(* CoDeSys 2.3 export: OSCAT260.TXT *)
(* Libraries: STANDARD.LIB 4.10.05 11:14:46 *)

(* Global variable list: Constants *)
VAR_GLOBAL CONSTANT
	(* setup Parameters *)
	STEP7 : BOOL := FALSE;

	(* Mathematische Konstanten *)
	PI1 : REAL := 3.14159265358979323846264338327950288;	(* Kreiszahl PI *)
	PI2 : REAL := 6.283185307179586476;					(* PI * 2 *)
	E : REAL := 2.71828182845904523536028747135266249;	(* Eulersche Konstante *)

	(* Physikalische Konstanten *)
	C0 : REAL := 299792458 ;							(* Lichtgeschwindigkeit in m/s *)
	EL : REAL := 1.60217653E-19;						(* elementarladung in Colomb = A * s *)
	GN : REAL := 9.80665; 								(* Erdbeschleunigung in m / s² *)
	TK : REAL := -273.15;									(* absoluter Nullpunkt in °C *)
	RU : REAL := 8.314472; 								(*Universelle Gaskonstante in J / (mol · K) *)
	PN : REAL := 101325;									(* NormalDruck in Pa *)

END_VAR

VAR_GLOBAL
END_VAR

(* revisionhistory
hm 3.3.2007
	extended accuracy of pi2
	renamed T0 to Tk for better compatibility with other libraries
	renamed C t0 c0 for better compatibility

hm	2.5.2007
	added RU universal gas constant

hm	1. oct 2007
	added setup parameter STEP7

hm 31. oct 2007
	added PN
*)

(* Data type *)
TYPE esr_data :
STRUCT
	typ : BYTE;
	adress : STRING(10);
	DS : DT;
	TS : TIME;
	data : ARRAY[0..7] OF BYTE;
END_STRUCT
END_TYPE

(* Data type *)
TYPE vector_3 :
STRUCT
	X : REAL;
	Y : REAL;
	Z : REAL;
END_STRUCT
END_TYPE

(* POU Building/actuators/actuator_2P, ST *)
FUNCTION_BLOCK actuator_2P
VAR_INPUT
	val : REAL;
	force : BOOL;
	force_in : BOOL;
END_VAR
VAR_INPUT CONSTANT
	self_act_time : TIME := t#10d;
	self_act_cycles : INT := 5;
	cycle_time : TIME := t#10m;
	min_ontime : TIME := t#10s;
	min_offtime : TIME := t#10s;
END_VAR
VAR_OUTPUT
	out :BOOL;
	pos : REAL;
END_VAR
VAR
	last_activation : TIME;
	count : INT;
	TON : TIME;
	tx : TIME;
	tc : TIME;
END_VAR


(*
version 1.5	27 dec 2007
programmer 	hugo
tested by		tobias

this is an intelligent actuator interface for any 2point actuator like coil drive.
the 2Point actuator can only switch on/off and therefore a input must be converted to on/off cycles.
the interface can be programmed with double click on the symbol for duty cyle, min_ontime and min_offtime to avoid flickering of the valve or flap.
in addition a self_act_time and self_act_cycles ca be programmed to switch n times on/off every self_act_time to avoid a valve to freeze.
a on and off input can be used to force the valve on or off at all times.
a additional pos output will always indicate the current position of a valve.
the input value must be between 0 and 1.

val		force	force_in	pos	out			
X		0		-			X		duty cycle X
-		1		1			1		1
-		1		0			0		0

*)
(* read system Time *)
tx := DWORD_TO_TIME(T_PLC_MS());
tc := tx - last_activation;

(* verify input to be between 0 and 1 *)
val := LIMIT(0,val,1);

(* check for min ontime or min offtime and wait if not passed *)
IF (out AND tc < min_ontime) OR (NOT out AND tc < min_offtime) THEN RETURN;

(* when force off then shutoff valve *)
ELSIF force AND NOT force_in THEN
	pos := 0;
	out := 0;
	last_activation := tx;
	count := 0;

(* if force on then turn on valve *)

ELSIF force AND force_in THEN
	pos := 1;
	out := 1;
	last_activation := tx;
	count := 0;

(* if nothing happened for self_act_time then do self activation cycles *)
ELSIF (tc >= self_act_time AND count = 0 AND self_act_cycles > 0) OR (count > 0 AND count < self_act_cycles * 2) THEN
	out := NOT out;
	last_activation := tx;
	count := count + 1;
	RETURN;
ELSIF count > 0 THEN
	count := 0;
ELSE
	ton := multime(cycle_time,val);
	IF ton < min_ontime / 2 THEN ton := t#0s; ELSIF ton < min_ontime THEN ton := min_ontime; END_IF;
	IF ton > cycle_time - min_offtime / 2 THEN ton := cycle_time; ELSIF ton > cycle_time - min_offtime THEN ton := cycle_time - min_offtime; END_IF;
	IF ton = t#0s THEN
		IF out =0 THEN
			pos := 0;
			RETURN;
		ELSE
			out := 0;
			pos := 0;
			last_activation := tx;
		END_IF;
	ELSIF ton = cycle_time THEN
		IF out = 1 THEN
			pos := 1;
			RETURN;
		ELSE
			out := 1;
			pos := 1;
			last_activation := tx;
		END_IF;
	END_IF;
	pos := TIME_TO_REAL(ton) / TIME_TO_REAL(cycle_time);
	(* output pulse generation *)
	IF out AND tc >= ton THEN
		out := 0;
		last_activation := tx;
	ELSIF NOT out AND tc >= cycle_time - ton THEN
		out := 1;
		last_activation := tx;
	END_IF;
END_IF;


(*
revision history:

hm		7.10.2006 		rev 1.1
	changed error pos could not reach 1 or 0 under certain conditions due to error in code.
	changed on and off in force and force_in for better usability.

hm		17.1.2007		rev 1.2
	deleted unused variable time_overflow

hm		15.9.2007		rev 1.3
	replaced time() with T_PLC_MS for compatibility and performance reasons

hm		19. 11 2007		rev 1.4
	replaced left over statement time() with tx

hm		27. 12. 2007	REV 1.5
	CHANGED CODE FOR BETTER PERFORMANCE
*)
END_FUNCTION_BLOCK

(* POU engineering/measurements/cycle_time, ST *)
FUNCTION_BLOCK cycle_time
VAR_INPUT
	rst : BOOL;
END_VAR
VAR_OUTPUT
	ct_min : TIME := t#0s;
	ct_max : TIME := t#0s;
	ct_last : TIME;
	systime : TIME;
	sysdays : INT;
	cycles : DWORD;
END_VAR
VAR
	last_cycle : TIME;
	tx: TIME;
	init: BOOL;
END_VAR


(*
	version 1.2	16 sep 2007
	programmer 	hugo
	tested BY		hans

this function block measures the cycle time and displays the last, min and max cycle time of the current task.
the resolution is 1ms.
the cycles output is a dword counter which counts the cycles.
a rst pulse on the input will reset all data.


*)
tx := DWORD_TO_TIME(T_PLC_MS()) - last_cycle;
IF rst THEN
	ct_min := t#10h;
	ct_max := t#0ms;
	cycles := 0;
ELSIF last_cycle > t#0s THEN
	IF tx < ct_min THEN ct_min := tx;
	ELSIF tx > ct_max THEN ct_max := tx;
	END_IF;
	ct_last := tx;
ELSIF ct_min = t#0s THEN
	ct_min := t#0s - t#1ms;
END_IF;
IF init THEN
	systime := systime + tx;
		IF systime >= t#1d THEN
			systime := systime - t#1d;
			sysdays := sysdays + 1;
		END_IF;
END_IF;
init := TRUE;
last_cycle := last_cycle + tx;
cycles := cycles + 1;

(*	revision history
hm 12.12.2006		rev 1.1
	added cycles output, a dword cycle counter.
hm 10.3.2007			rev 1.2
	changed initialization of ct_min to t#10h for compatibility with siemens s7

hm	16.9.2007		rev 1.2
	changed Time() in T_PLC_MS() for compatibility resons

*)
END_FUNCTION_BLOCK

(* POU engineering/measurements/T_PLC_MS, ST *)
FUNCTION T_PLC_MS : DWORD
VAR CONSTANT
	debug : BOOL := FALSE;
	N : INT := 0;
	offset : DWORD := 0;
END_VAR
VAR
	tx : TIME;
	temp : DWORD := 1;
END_VAR

(*
version 1.1	12 nov 2007
programmer 	hugo
tested by		tobias

T_PLC_MS reads the internal PLC timer and return the time, it has the advantage to be able to set a debug mode 
and speed up the counter to test the plc timer overrun which occurs every 50 days respectively 25 days at siemens S7
this routine also allows to correct the behavior of s7 where the internal plc counter will not count all 32 bits.

*)
tx := TIME();
T_PLC_MS := TIME_TO_DWORD(Tx);
(* hier muss die korrektur für step7 stattfinden
plctime muss den vollen wertebereich von time ausnutzen:
wenn bei step7 time -24tage bis plus 24 tage ist dann muss der timer auch beim überlauf auf -24tage springen 
und auf keinen fall auf 0 !!!!
für siemens muss ein weiterer fb im main eingebunden werden der sicherstellt das alle 32 bits durchgezählt werden.
es kann nur ein fb sein den er muss sich das oberste (32te) bit merken.
oder etwa spring s7 bei überlauf auf -24 tage????? dann wäre keine korrektur nötig.
*)
IF debug THEN
	T_PLC_MS := (SHL(T_PLC_MS,N) OR SHL(temp,N)-1) + Offset;
END_IF;

(* revision history
hm	14.9.2007	rev 1.0
	original version

hm	12. nov 2007	rev 1.1
	added temporaray variable tx because some compilers could not handle time() as an argument

*)
END_FUNCTION

(* POU engineering/signal processing/Offset, ST *)
FUNCTION Offset : REAL
VAR_INPUT
	X : REAL;
	O1, O2, O3, O4 : BOOL;
	D : BOOL;
END_VAR
VAR_INPUT CONSTANT
	Offset_1 : REAL;
	Offset_2 : REAL;
	Offset_3 : REAL;
	Offset_4 : REAL;
	default : REAL;
END_VAR

(*
version 1.0	12 jan 2007
programmer 	oscat
tested by		tobias

The Function offset adds offsets to an analog signal depending on digital inputs.
all selected offsets are added at the same time.
with the input D a default value instead of the input X can be used.

*) 
IF D THEN Offset := default; ELSE Offset := X; END_IF;
IF O1 THEN Offset := Offset + offset_1; END_IF;
IF O2 THEN Offset := Offset + offset_2; END_IF;
IF O3 THEN Offset := Offset + offset_3; END_IF;
IF O4 THEN Offset := Offset + offset_4; END_IF;
END_FUNCTION

(* POU Time&Date/multime, ST *)
FUNCTION multime : TIME
VAR_INPUT
	t : TIME;
	M : REAL;
END_VAR
VAR
END_VAR


(*
version 1.0	2 oct 2006
programmer 	hugo
tested by		tobias

multiplies a time by a real number and returns a time
*)
multime := REAL_TO_TIME(TIME_TO_REAL(t)*M);
END_FUNCTION

(* POU Building/actuators/actuator_3P, ST *)
FUNCTION_BLOCK actuator_3P
VAR_INPUT
	in : REAL;
	force : BOOL;
	on : BOOL;
	end_pos : BOOL;
	diag : BOOL;
END_VAR
VAR_INPUT CONSTANT
	min_ontime : TIME := t#10s;
	min_offtime : TIME := t#10s;
	max_runtime : TIME := t#60s;
	auto_diag_time : TIME := t#10d;
	cal_runtime : TIME := t#600s;
	switch_available: BOOL;
END_VAR
VAR_OUTPUT
	out1 : BOOL;
	out2 : BOOL;
	pos : REAL;
	busy : BOOL;
	error : BOOL;
END_VAR
VAR
	val: REAL;
	tx : TIME;
	last_diag: TIME;
	last : TIME;
	runtime_1 : TIME;
	runtime_2 : TIME;
	state : INT;
	rout: FT_rmp;
	end : R_TRIG;
	cal_timer: TIME;
	Tn: TIME;
END_VAR


(*
version 1.3	 15 sep 2007
programmer 	hugo
tested by		tobias

actuator_3P is an interface for a 3 point actuator.
a 3P actuator is a motor with 2 directions that drives a valve or flap. the position of the valve or flap is controlled by runtime of the motor foreward or backward.
the available inputs are:
in is a real value which specifies the position of the actuator, 0 = 0% and 1 = 100% any value <0 or > 1 is limited to 0 or 1.
a force input must be low for normal operation and if switched high, the motor can only be controlled for 0% or 100% positions with the on input.
an and pos input is available for a end_pos switch, this switch indicates the valve or flap to be at either 0% or 100%
a diag input can at any time start a diag cycle which turns the motor towards the 0% position, then measures the runtime to 100% and then the runtime to 0%
these runtimes are stored and used for absolute positioning of the motor during normal operation.
a setup constand "auto_diag_time can be used to specify how often the actuator repeates this auto_diag cycla automatically.
at power on a cycle is perfomed automatically.
a 0 for this value means auto diag is never performed.

the outputs ar out1 and out2 for up and down direction of the motor. to avoid flickering the output can be programmed for min_ontime and min_offtime.
a pos outout indicates the absulute position of the actuator during operation and a busy output indicates the actuator is busy.
a error output is initiated when the specified max_runtime is reached by any direction during debug.
also when the up and down direction differs by more then 10% the error output is set.

for absolute positioning accuracy the actuator has a setup variable "cal_runtime" if this is set the actuator measures the total runtime of the motors and when this 
cal_runtime is exceeded it resets the actuator to 0% position and sets the output again to assure absolute accuracy.

autodiag and calibration can be shut off by setting the appropriate values to 0.
a switch_available setup variable specifies if end_pos switches are available.

*)
(* setup *)
Tn := DWORD_TO_TIME(T_PLC_MS());
tx := Tn - last;
end(clk := end_pos);

(* init only when first started *)
IF state = 0 THEN
	runtime_1 := max_runtime;
	runtime_2 := max_runtime;
	state := 1;
	rout(KR := 1000 / TIME_TO_REAL(runtime_1), KF := 1000 / TIME_TO_REAL(runtime_1) );
	tx := t#0s;
	last := Tn;
	last_diag := last;
END_IF;

(* check for end_sw and stop if reached *)
IF switch_available AND out1 AND end.Q THEN
	(* upper limit has been reached *)
	out1 := 0;
	rout(rmp := 0, in := 1);
	rout.Rmp := 1;
ELSIF switch_available AND out2 AND end.Q THEN
	(* lower limit has been reached *)
	out2 := 0;
	rout(rmp := 0, in := 0);
	rout.Rmp := 1;
END_IF;

(* check for min_offtime and min_ontime and return if it has not elapsed *)
IF NOT busy AND tx < min_offtime THEN RETURN;
ELSIF busy AND tx < min_ontime THEN RETURN;

(* check for last diag cycle and start diag if auto_diag_time has elapsed *)
ELSIF (tn - last_diag > auto_diag_time AND state > 10 AND auto_diag_time > t#0s) OR (diag AND state >= 10) THEN state := 1;

(* check if force pin is high *)
ELSIF force THEN state := 10;

(* check if calibration is necessary *)
ELSIF cal_timer > cal_runtime AND state = 99 AND cal_runtime > t#0s THEN state := 20;
END_IF;

(* state machine for operation *)
CASE state OF

1 :	(* diagnostic start *)
	(* all data is reset and out2 is turned on to make sure we start from top position *)
	last_diag := tn;
	diag := 0;
	state := 2;
	pos := 0;
	busy := 1;
	last := tn;
	out1 := 0;
	out2 := 1;
	RETURN;

2:	(* wait for max_runtime or end_pos to be reached *)
	IF tx < max_runtime AND NOT end.Q THEN RETURN; END_IF;
	state := 3;
	last := tn;
	out1 := 1;
	out2 := 0;
	RETURN;

3: 	(* measure runtime_2 *)
	IF tx < max_runtime AND NOT end.Q THEN RETURN; END_IF;
	state := 4;
	runtime_1 := tx;
	last := tn;
	out1 := 0;
	out2 := 1;
	RETURN;

4:	(* measure runtime_1 *)
	IF tx < max_runtime AND NOT end.Q THEN RETURN; END_IF;
	state := 99;
	runtime_2 := tx;
	last := tn;
	out2 := 0;
	busy := 0;
	(* reset the output ramp generator to the 0% position as the valve is after diags *)
	rout(rmp := 0, in := 0);
	rout.Rmp := 1;
	cal_timer := t#0s;
	IF differ(TIME_TO_REAL(runtime_1), TIME_TO_REAL(runtime_2), TIME_TO_REAL(max_runtime) * 0.1) THEN error := TRUE;
	ELSIF runtime_1 > multime(max_runtime, 0.9) AND switch_available THEN error := TRUE;
	ELSIF runtime_2 > multime(max_runtime, 0.9) AND switch_available THEN error := TRUE;
	END_IF;
	RETURN;

10: (* force pin is active, outputs are forced on or off by the on pin *)
	IF on AND NOT out2 THEN val := 1;
	ELSIF NOT on AND NOT out1 THEN val := 0;
	END_IF;
	IF NOT force THEN state := 99; END_IF;

20 : (* calibrate to allow for correction of positioning error addig up *)
	cal_timer := t#0s;
	state := 21;
	pos := 0;
	busy := 1;
	last := tn;
	out1 := 0;
	out2 := 1;
	RETURN;

21:	(* after end_sw or max_runtime we can be sure to have reached the 0% position *)
	IF tx < max_runtime AND NOT end.Q THEN RETURN; END_IF;
	state := 99;
	out2 := 0;
	busy := 0;
	last := tn;
	rout(rmp := 0, in := 0);
	rout.Rmp := 1;
	RETURN;

99: (* normal operation *)
	(* only if input changes for an equivalent of min_ontime then change the output *)
	(* if there is a directional change then wait until last step is finished *)
	IF in < TIME_TO_REAL(min_ontime)/TIME_TO_REAL(max_runtime)/2 THEN val := 0;
	ELSIF in > 1 - TIME_TO_REAL(min_ontime)/TIME_TO_REAL(max_runtime)/2 THEN val := 1;
	ELSIF differ(LIMIT(0,in,1), val, TIME_TO_REAL(min_ontime) / TIME_TO_REAL(max_runtime)) OR in = 0 OR in = 1 THEN
		IF in < val AND NOT out1 THEN val := in;
		ELSIF in > val AND NOT out2 THEN val := in;
		END_IF;
	END_IF;

END_CASE;

(* output ramp generator *)
rout(in := val);
out1 := rout.busy AND rout.UD;
out2 := rout.busy AND NOT rout.UD;
pos := rout.out;

(* set the busy output and if busy goes low, then set the last time in order to check for min_offtime *)
IF NOT busy AND rout.busy THEN
	last := tn;
ELSIF busy AND NOT rout.busy THEN
	cal_timer := cal_timer + tx;
	last := tn;
END_IF;
busy := rout.busy;



(* revision history

19.10.2006	rev 1.1
	added security checks for end_switch to avoid overrun of the end_switch, hans

23.1.2007		rev 1.2
	deleted unused variables force_on and force_off

15.9.2007	hm	rev 1.3
	replaced Time() with T_PLC_MS for compatibility and performance reasons

*)
END_FUNCTION_BLOCK

(* POU mathematical/functions/FT_rmp, ST *)
FUNCTION_BLOCK FT_rmp
VAR_INPUT
	Rmp : BOOL := TRUE;
	in : REAL;
	KR : REAL;
	KF : REAL;
END_VAR
VAR_OUTPUT
	out : REAL;
	busy : BOOL;
	UD : BOOL;
END_VAR
VAR
	tx: TIME;
	last: TIME;
	init: BOOL;
END_VAR

(*
	version 1.3	17 sep 2007
	programmer 	oscat
	tested BY		oscat

this ramp function follows an input signal with a linear ramp up or down, the up or down speed can be set with KF and KR.
a K factor of 1 means 1 unit per second on the output. K factors can only be positive and not negative.
a busy output signals the ramp is running or busy false means the in value is present on the output.
a rmp input false means the output follows the input dierctly while a rmp = true means the output follows the input with a ramp.
a updn output signal the directon of the ramp (up or down).

*)
(* read system time *)
tx := DWORD_TO_TIME(T_PLC_MS()) - last;

IF NOT init THEN
	init := TRUE;
	last := tx;
	tx := t#0s;
	out := in;
END_IF;
IF NOT rmp THEN
	out := in;
	busy := FALSE;
ELSIF out > in AND kf > 0 THEN
	(* ramp down *)
	out := out - TIME_TO_REAL(tx) / 1000 * KF;
	IF out < in THEN out := in; END_IF;
ELSIF out < in AND kr > 0 THEN
	(* ramp up *)
	out := out + TIME_TO_REAL(tx) / 1000 * KR;
	IF out > in THEN out := in; END_IF;
END_IF;

(* set busy and dir flags *)
IF out < in THEN
	busy := TRUE;
	ud := 1;
ELSIF out > in THEN
	busy := TRUE;
	ud := 0;
ELSE
	busy := FALSE;
END_IF;
last := last + tx;


(* revision history:

hm 8.10.2006			rev 1.1
	added ud output

hm 12. feb 2007		rev 1.2
	added init variable and corrected a possible startup problem

hm	17. sep 2007	rev 1.3
	replaced time() with t_plc_ms() for compatibility reasons

*)
END_FUNCTION_BLOCK

(* POU mathematical/differ, ST *)
FUNCTION differ : BOOL
VAR_INPUT
	in1 : REAL;
	in2 : REAL;
	X : REAL;
END_VAR
VAR
END_VAR

(*
version 1.0	8 oct 2006
programmer 	hugo
tested by		tobias

this function checks if in1 differs more then x from in2
the output is true if in1 < in2 - x or in1 > in2 + X
*)
differ := in1 < in2 - X OR in1 > in2 + X;
END_FUNCTION

(* POU Building/actuators/actuator_pump, ST *)
FUNCTION_BLOCK actuator_pump
VAR_INPUT
	in : BOOL;
	manual : BOOL;
	rst : BOOL := FALSE;
END_VAR
VAR_INPUT CONSTANT
	min_ontime : TIME := t#10s;
	min_offtime : TIME := t#10s;
	run_every : TIME := t#10000m;
END_VAR
VAR_OUTPUT
	pump : BOOL;
	runtime : REAL;
	cycles : REAL;
END_VAR
VAR
	tx : TIME;
	last_change : TIME;
	meter : ontime;
	old_man : BOOL;
	init: BOOL;
END_VAR

(*
	version 1.2	15 sep 2007
	programmer 	oscat
	tested BY		oscat

actuator_pump is a pump interface which can be controlled by an input in and an input manual.
in or manual high turns the pump output on.
a rst input is used to reset the runtime counters.
when the pump was not active for a time run_every the actuator turns on the pump automatically for min_ontime.
two setup variables min_ontime and min_offtime guarantee a minimum runtime and offtime of the pump.
the units are hours and the output type is real to prevent from overfow.

*)
tx := DWORD_TO_TIME(T_PLC_MS());

IF NOT init THEN
	init := 1;
	last_change := tx;
ELSIF rst THEN
	rst := FALSE;
	meter(rst := 1);
	meter.rst := 0;
ELSIF manual AND NOT pump AND NOT old_man THEN
	last_change := tx;
	pump := 1;
ELSIF NOT manual AND old_man AND pump AND NOT in THEN
	last_change := tx;
	pump := 0;
ELSIF in AND NOT pump AND tx - last_change >= min_offtime THEN
	last_change := tx;
	pump := 1;
ELSIF pump AND NOT in AND NOT manual AND tx - last_change >= min_ontime THEN
	last_change := tx;
	pump := 0;
ELSIF NOT pump AND tx - last_change >= run_every THEN
	last_change := tx;
	pump := 1;
END_IF;

meter(in := pump);
runtime := meter.ontime;
cycles := meter.cycles;
old_man := manual;

(*
27.12.2006	rev 1.1	hm
	fixed a failure while the pump would run for tmin after startup.

15.9.2007	hm	rev 1.2
	replaced Time() with T_PLC_MS for compatibility and performance reasons

*)
END_FUNCTION_BLOCK

(* POU engineering/measurements/Meter, ST *)
FUNCTION_BLOCK Meter
VAR_INPUT
	M1, M2 : REAL;
	I1, I2 : BOOL;
	D : REAL := 1;
	RST : BOOL;
END_VAR
VAR_OUTPUT RETAIN
	MX : REAL;
END_VAR
VAR
	int1 : FT_INT;
	int2 : FT_INT;
END_VAR

(*
	version 1.0	16 sep 2007
	programmer 	oscat
	tested BY		oscat

METER measures usage of power or similar values the output MX is the summ of the inputs over time.
MX := sum over time of I1 * P1 + I2 * P2.
a simple example is the consumption counter for a 2 stage oil burner where stage 1 is 10KW and stage 2 is 20KW.
I1 and I2 decide which value is accounted for, I1 = True only counts P1, I2 is True counts P2 
and I1 and I2 is true counts P1 and P2.
the meter can be used for all kind of consumption meters. P1 and P2 can change on the fly.

*)
int1(in := M1, Run := I1, RST := RST, out_min := -1E-38, out_max :=3E+38);
int2(in := M2, Run := I2, RST := RST, out_min := -1E-38, out_max :=3E+38);
MX := (int1.Out + int2.Out) / D;

(* revision history

hm	7.2.2007		rev 1.0
	original version

*)
END_FUNCTION_BLOCK

(* POU engineering/control/FT_INT, ST *)
FUNCTION_BLOCK FT_INT
VAR_INPUT
	in : REAL;
	K : REAL := 1;
	run : BOOL := 1;
	rst: BOOL := 0;
	out_min : REAL := -1000;
	out_max : REAL := 1000;
END_VAR
VAR_OUTPUT
	Out : REAL;
	ET: TIME;
END_VAR
VAR
	last: DWORD;
	in_last : REAL;
	tx: DWORD;
	init: BOOL;
	tc: DWORD;
	eti : DWORD;
END_VAR


(*
version 1.5	2 dec 2007
programmer 	hugo
tested by		tobias

FT_int is an integrator with input IN and factor K.
integration is only done while run = true, if run is false integration is stopped and the out remains at the last value.
if run is left unconnected, run is considered true by the function block.
the output ET will display the total integration time from last reset.
a rst input will reset output and the timer ET to 0.
the out_min and out_max values can be set to ,imit the output value range. 
out _min is preset to -1000 and out_max is preset to 1000.
the default for K is 1.

 
*)
(* read and store system time *)
tx := T_PLC_US();
tc := tx - last;

(* startup initialisation *)
IF rst OR NOT init THEN
	out := 0;
	ET := t#0s;
	init := TRUE;
	last := tx;
ELSIF run AND tc > 0 THEN
	last := tx;
	out := LIMIT(out_min, out + (in + in_last) * tc * K / 2000000, out_max);
	eti := eti + tc;
	et := DWORD_TO_TIME(eti / 1000);
ELSIF NOT run THEN
	last := tx;
END_IF;
in_last := in;

(*
hm 13.12.2006	rev 1.1
	changed to "trapezregel" which increases accuracy
	before out := out + in * time new: out := out + (in + in_last) / 2 * time

hm 15.1.2007		rev 1.2
	added default for k to be 1.

hm	15.9.2007		rev 1.3
	replaced time() with T_PLC_US for compatibility and performance reason
	increased internal accuracy to microseconds

hm 29. oct 2007		rev 1.4
	changed code so int will not be called is time difference is 0 to increase accuracy on systems
	with cycle times below 1ms

hm	2. dec 2007	 	rev 1.5
	changed code for better performance
*)
END_FUNCTION_BLOCK

(* POU engineering/measurements/T_PLC_US, ST *)
FUNCTION T_PLC_US : DWORD
VAR CONSTANT
	debug : BOOL := FALSE;
	N : INT := 0;
	offset : DWORD := 0;
END_VAR
VAR
	tx : TIME;
	temp : DWORD := 1;
END_VAR

(*
version 1.1	12 nov 2007
programmer 	hugo
tested by		tobias

T_PLC_US reads the internal PLC timer and return the time, it has the advantage to be able to set a debug mode 
and speed up the counter to test the plc timer overrun which occurs every 50 days respectively 25 days at siemens S7
this routine also allows to correct the behavior of s7 where the internal plc counter will not count all 32 bits.

*)
tx := TIME();
T_PLC_US := TIME_TO_DWORD(Tx)*1000;
(* hier muss die korrektur für step7 stattfinden
plctime muss den vollen wertebereich von time ausnutzen:
wenn bei step7 time -24tage bis plus 24 tage ist dann muss der timer auch beim überlauf auf -24tage springen 
und auf keinen fall auf 0 !!!!
für siemens muss ein weiterer fb im main eingebunden werden der sicherstellt das alle 32 bits durchgezählt werden.
es kann nur ein fb sein den er muss sich das oberste (32te) bit merken.
oder etwa spring s7 bei überlauf auf -24 tage????? dann wäre keine korrektur nötig.
*)
IF debug THEN
	T_PLC_US := (SHL(T_PLC_US,N) OR SHL(temp,N)-1) + Offset;
END_IF;

(* revision history
hm	14.9.2007	rev 1.0
	original version

hm	12. nov 2007	rev 1.1
	added temporaray variable tx because some compilers could not handle time() as an argument

*)
END_FUNCTION

(* POU engineering/measurements/ontime, ST *)
FUNCTION_BLOCK ontime
VAR_INPUT
	in : BOOL;
	rst : BOOL := FALSE;
END_VAR
VAR_OUTPUT RETAIN
	ontime : REAL;
	last_on : REAL;
	cycles : REAL;
END_VAR
VAR
	tx: DWORD;
	last : DWORD;
	edge : BOOL := 0;
	L_time1, H_time1, L_time2, H_time2 : DWORD;
	temp: DWORD;
END_VAR

(*
version 1.4	2 dec 2007
programmer 	oscat
tested by		tobias

M_runtime measures the ontime of a signal in hours.
the output is of type real because the time type will overflow within 49 days.
the units are hours.

*)
(* read system time *)
tx := T_PLC_MS();

IF rst THEN
	L_time1 := 0;
	H_time1 := 0;
	cycles := 0;
	L_time2 := 0;
	H_time2 := 0;
	ontime := 0;
	last_on := 0;
ELSIF in THEN
	temp := L_time1;
	L_time1 := L_time1 + (tx-last);
	IF temp > L_time1 THEN H_time1 := H_time1 + 1; END_IF;
	ontime := L_time1/3600000.0 + 1193.046471 * H_time1;
	temp := L_time2;
	L_time2 := L_time2 + (tx-last);
	IF temp > L_time2 THEN H_time2 := H_time2 +2; END_IF;
	last_on := L_time2/3600000.0 + 1193.046471 * H_time2;
	IF NOT edge THEN
		cycles := cycles +1;
		last_on := 0;
		L_time2 := 0;
		H_time2 := 0;
	END_IF;
END_IF;
last := tx;
edge := in;

(* revision history
hm 22.2.2007		rev 1.1
	changed VAR RETAIN PERSISTENT to VAR RETAIN for better compatibility
	wago lon contollers do not support persisitent

hm 2.8.2007		rev 1.2
	adding time up in a real number will automatically lead to the point where 
	small time scales like the cycle time will be below the resolution of real and therefore
	ontime would not increase in small steps as necessary
	the time is now measured internally in two  dwords and be converted to real only for
	output purposes.
	deleted the variable power because it was unnecessary

hm	16.9.2007	rev 1.3
	changes time() to T_plc_ms() for compatibility reasons

hm	2. dec. 2007	rev 1.4
	chaged code for better performance
*)
END_FUNCTION_BLOCK

(* POU Building/actuators/actuator_UD, ST *)
FUNCTION_BLOCK actuator_UD
VAR_INPUT
	UD : BOOL;
	ON : BOOL;
	Manual : BOOL := 0;
	Up : BOOL;
	Dn : BOOL;
	off : BOOL := 0;
	YUP_in : BOOL;
	YDN_in : BOOL;
END_VAR
VAR_INPUT CONSTANT
	TON : TIME;
	TOFF : TIME;
	out_return : BOOL;
END_VAR
VAR_OUTPUT
	Yup : BOOL;
	Ydn : BOOL;
	status : BYTE;
END_VAR
VAR
	tx : TIME;
	last : TIME;
	init: BOOL;
END_VAR

(*
version 1.2	15 sep 2007
programmer 	hugo
tested by		tobias

out_ud is a up/dn or Right/left locked output driver.
it can be controlled by automatic inputs UD and ON as well as manual inputs for up and dn.
a security input to shut off at any time is prvided by the off input.
two time set inputs ton and toff specify a minimum on time for outputs and a minimum off time before the next output can become active.
the module assures that only one output can be active at any time.
for higher security pls make sure you use hardware locking of the outputs to prevent from defective wiring or outputs.
further security is provided b feedback inputs Yup_in and Ydn_in which are separate inputs for the output signal, if these inputs are not available 
pls connect them directly to Yup and Ydn.
manual mode will override automatic mode by setting the manual input high.
a status output will be 0 for normal operation or 1 - 99 for error reporting and 101 - 199 for status reporting
The status output is ESR comptible.
*)
(* read system time *)
tx := DWORD_TO_TIME(T_PLC_MS());

IF NOT init THEN
	(* INITIALIZATION AT FIRST CALL *)
	last := tx;
	init := TRUE;
ELSIF off THEN
	(* emergency shut off detected *)
	Yup := FALSE;
	Ydn := FALSE;
	last := tx;
	status := 101;

(* WATH FOR MIN TON TIME *)
ELSIF ((Yup OR Ydn) AND tx - last < Ton) THEN RETURN;
ELSIF NOT yup AND NOT ydn AND tx - last < toff THEN	RETURN;

(* manual operation *)
ELSIF manual THEN
	status := 102;
	(* directional chage set both outs 0 first *)
	IF yup AND NOT up OR ydn AND NOT dn THEN
		ydn := 0;
		yup := 0;
		last := tx;
	(* manual up operation *)
	ELSIF UP AND NOT DN AND NOT OFF THEN
		Ydn := 0;
		Yup := 1;
		last := tx;
		status := 103;
	(* manual down operation *)
	ELSIF DN AND NOT UP AND NOT OFF THEN
		Yup := 0;
		Ydn := 1;
		last := tx;
		status := 104;
	(* maual mode but no up or down *)
	ELSE
		IF YUP OR YDN THEN LAST := tx; END_IF;
		Yup := 0;
		Ydn := 0;
	END_IF;

(* automatic operation *)
ELSE
	(* directional change set outputs low first *)
	IF yup AND NOT ud OR ydn AND UD THEN
		yup := 0;
		ydn := 0;
		last := tx;
	(* automatic up operation *)
	ELSIF Ud AND on AND NOT OFF THEN
		Ydn := 0;
		Yup := 1;
		last := tx;
		status := 111;

	(* automatic down operation *)
	ELSIF NOT UD AND on AND NOT OFF THEN
		Yup := 0;
		Ydn := 1;
		last := tx;
		status := 112;
	(* standby mode *)
	ELSE
		IF Yup OR Ydn THEN last := tx; END_IF;
		Yup := 0;
		Ydn := 0;
		status := 110;
	END_IF;
END_IF;

(* make sure Yup and Ydn are never on at the same time *)
IF Ydn AND Yup_in AND out_return THEN
	Ydn := 0;
	status := 1;
END_IF;
IF Yup AND Ydn_in AND out_return THEN
	Yup := 0;
	status := 2;
END_IF;

(* revision history
hm 22. jan 2007	rev 1.1
	added status output
	changed inputs ton, toff to config variables
	added config var out_return to enable yup_in and Ydn_in
	manual mod will override automatic mode 

hm	15.9.2007	rev 1.2
	replaced Time() with T_PLC_MS for compatibility and performance reasons
*)
END_FUNCTION_BLOCK

(* POU Building/electrical/click, ST *)
FUNCTION_BLOCK click
VAR_INPUT
	in : BOOL;
END_VAR
VAR_OUTPUT
	Q : BOOL;
	single : BOOL;
	double : BOOL;
	triple : BOOL;
	status: BYTE;
END_VAR
VAR_INPUT CONSTANT
	T_debounce : TIME := t#10ms;
	T_short : TIME := t#200ms;
	T_pause : TIME := t#500ms;
	T_reconfig : TIME := t#1m;
END_VAR
VAR
	debounce : TON;
	tx : TIME;
	last : TIME;
	init : BOOL;
	edge : BOOL;
	standby: BOOL;
	state: INT;
END_VAR

(*
version 1.2	15 sep 2007
programmer 	oscat
tested by		tobias

click checks an input for single, double or tripple click and sets the corresponding output single, doulbe or triple for the time the input stays high at the last click.
the maximum high and low time for a click can beconfigrured with setup variables.
the input cinfigures itself to be high or low active dependung on which state the input stays longer than t_reconfig.

*)
(* read system time *)
tx := DWORD_TO_TIME(T_PLC_MS());

(* set last and tx if never started before *)
IF NOT init THEN
	init := TRUE;
	last := tx;
	debounce.PT := T_debounce;
	standby := in;
END_IF;

(* debounce input *)
debounce(in := in XOR standby);
Q := debounce.Q;

(* delete outputs if input is inactive *)
IF NOT Q THEN
	single := FALSE;
	double := FALSE;
	triple := FALSE;
	status := 110;
END_IF;

(* check for input edge *)
IF Q XOR edge THEN
	edge := in;
	last := tx;
	IF Q THEN state := state + 1; END_IF;
END_IF;

IF (q AND tx - last >= T_short) OR (NOT q AND tx - last >= t_pause) THEN
	CASE state OF
		1:	single := TRUE;
			status := 111;
		2:	double := TRUE;
			status := 112;
		3:	triple := TRUE;
			status := 113;
	END_CASE;
	state := 0;
END_IF;

(* determine if high or low active *)
IF tx - last >= t_reconfig THEN
	standby := in;
	last := tx;
END_IF;



(* revision history

15 Feb 2007	rev 1.0	hm
	created original version

18.5.2007		rev 1.1 hm
	corrected an error while execution would stop after t_reconfig elapsed.

15.9.2007		rev 1.2 hm
	replaced Time() with T_PLC_MS for compatibility and performance reasons

*)
END_FUNCTION_BLOCK

(* POU Building/electrical/dimm_i, ST *)
FUNCTION_BLOCK dimm_i
VAR_INPUT
	set : BOOL;
	in : BOOL;
	rst : BOOL;
END_VAR
VAR_INPUT CONSTANT
	T_debounce : TIME := T#10ms;
	T_reconfig : TIME := T#10s;
	T_on_max : TIME := T#0h;
	T_dimm_start : TIME := T#1s;
	T_dimm: TIME := T#3s;
END_VAR
VAR_OUTPUT
	Q : BOOL := 0;
	out : BYTE := 0;
END_VAR
VAR
	tx : TIME := T#0s;
	last_edge : BOOL;
	state : BYTE := 0;
	edge : BOOL := 0;
	r_edge : BOOL := 0;
	T_on : TIME;
	dimm_up: BOOL;
	last_step : TIME;
	tn: TIME;
END_VAR

(*
version 1.3	15 sep 2007
programmer 	hugo
tested by		tobias

this is an intelligent dimmer interface with an autoset feature for "in" it will automatically detect the type of switch:
low active pulses or high high active pulses are allowd for in.
a configurable debounce timer will debounce input signals
if t_on_max is set to anything other then 0 the output will be turned off after the max on time is reached.
the times for debounce, dimming ramp, wait time before dimming and max on time are all programmable.

the dimmer has outputs Q for on and off and also out with the analog dimm value.

*)
(* read system time *)
tn := DWORD_TO_TIME(T_PLC_MS());;

IF rst THEN
	state := 0;
	Q := 0;
	dimm_up := TRUE;
ELSIF set THEN
	state := 0;
	Q := TRUE;
	out := 255;
	dimm_up := FALSE;
	T_on := Tn;
ELSE
	CASE state OF
	(* state 0 wait for activity *)
	0 :	IF (r_edge AND in AND NOT edge) OR (NOT r_edge AND NOT in AND edge) THEN
			IF t_debounce = t#0s THEN state := 2;  ELSE state := 1; END_IF;
			tx := Tn;
			last_edge := in;
		END_IF

	(* state 1 debouncing *)
	1:	IF Tn - T_debounce >= tx THEN
			state := 2;
			tx := Tn;
		END_IF;

	(* state 2 wait for second edge to toggle output *)
	2:	IF Tn - T_dimm_start >= tx THEN
			state := 3;
			tx := Tn;
			(* time to switch elapsed without switching if Q = 0 turn on output and start dimming at 1 *)
			IF NOT Q THEN
				Q := TRUE;
				t_on := tx;
				out := 1;
				dimm_up := TRUE;
			ELSE
				IF out =255 THEN dimm_up := FALSE; END_IF;
			END_IF;
		ELSIF in XOR edge THEN
			(* wait for edge to toggle output and stop all activity *)
			IF Q THEN
				Q := FALSE;
				state := 0;
			ELSE
				Q := TRUE;
				state := 3;
				IF out = 0 THEN out := 255; END_IF
				IF out = 255 THEN dimm_up := FALSE; END_IF;
				tx := Tn;
				t_on := tx;
			END_IF;
		END_IF;

	(* state 3 entered dimming phase *)
	3:	IF in AND r_edge THEN
			(* generate ramp *)
			tx := Tn;
			IF tx >= last_step + T_dimm / 255 THEN
				last_step := tx;
				IF dimm_up AND out < 255 THEN
					out := out + 1;
					IF out = 255 THEN
						dimm_up := FALSE;
						state := 0;
					END_IF;
				ELSIF NOT dimm_up AND out > 0 THEN
					out := out -1;
					IF out = 0 THEN
						Q := FALSE;
						state := 0;
						dimm_up := TRUE;
					 END_IF;
				 END_IF;
			END_IF;
		ELSE
			dimm_up := NOT dimm_up;
			state := 0;
		END_IF;

	END_CASE;

	(* check for max t_on time and reset output if too long *)
	IF Q AND t_on_max > T#0s AND Tn - t_on_max >= T_on THEN Q := 0; END_IF;

	(* check for reconfig and set R_edge to high for rising edge sensitivity *)
	IF Tn - T_reconfig >= tx THEN R_edge := NOT in; END_IF;

	(* set edge to follow in for next edge detection *)
	edge := in;
END_IF;


(* revision history

hm 22.1.2007		rev 1.1
	deleted unused structure ramp

hm 2.feb 2007		rev 1.2
	changed structure to read time() at the beginning for better time consistency if a higher priorized tak interrupts dimm_i
	added statements in case structure for state 1 to allow for short 1 cycle input pulses

hm 	15.9.2007		rev 1.3
	replaced Time() with T_PLC_MS for compatibility and performance reasons

*)
END_FUNCTION_BLOCK

(* POU Building/electrical/F_Lamp, ST *)
FUNCTION_BLOCK F_Lamp
VAR_INPUT
	SWITCH : BOOL;
	DIMM : BYTE := 255;
	Rst : BOOL;
END_VAR
VAR_OUTPUT
	Lamp : BYTE;
	ontime : REAL;
	cycles : REAL;
	Status : BYTE;
END_VAR
VAR_INPUT CONSTANT
	T_no_Dimm : REAL := 100;
	T_Maintenance : REAL := 15000;
END_VAR
VAR
	runtime : ontime;
	maintenance: BOOL;
END_VAR

(*
version 1.1	8 Feb 2007
programmer 	hugo
tested by		tobias

F_Lamp is an interface to flourescent lamps. its main purpose is to protect flourescent lamps from dimming within the first T_NO_DIMM Time.
If Flourescent Lamps are dimmed during the first 100 hours the lifetime of the lamp is reduced dramatically.
The interface also counts ontime and cycles of the lamp for maintanance purposes.

*)
IF rst THEN
	runtime.rst := TRUE;
	runtime();
	runtime.rst := FALSE;
	ontime := runtime.ontime;
	cycles := runtime.cycles;
	maintenance := FALSE;
ELSE
	runtime(in := Switch);
	ontime := runtime.ontime;
	cycles := runtime.cycles;
END_IF;

IF NOT maintenance AND runtime.ontime >= T_maintenance AND T_Maintenance > 0 THEN
	status := 120;
	maintenance := TRUE;
ELSIF Switch THEN
	IF runtime.ontime < T_no_Dimm THEN
		Lamp := 255;
		STATUS := 111;
	ELSE
		Lamp := DIMM;
		status := 112;
	END_IF;
ELSE
	lamp := 0;
	status := 110;
END_IF;
END_FUNCTION_BLOCK

(* POU Building/electrical/Pulse_Length, ST *)
FUNCTION_BLOCK Pulse_Length
VAR_INPUT
	in : BOOL;
END_VAR
VAR_OUTPUT
	short : BOOL;
	middle : BOOL;
	long : BOOL;
END_VAR
VAR_INPUT CONSTANT
	T_short : TIME := t#100ms;
	T_long : TIME := t#1s;
END_VAR
VAR
	tx : TIME;
	tn: TIME;
	edge : BOOL;
END_VAR

(*
version 1.1	15 sep 2007
programmer 	oscat
tested by		tobias

Pulse_length indicates on 3 outputs if an input pulse had been shorter than T_short (short = True), longer than T_long (long = True) or between T_short and T_long (middle = True).

*)
(* read system time *)
tx := DWORD_TO_TIME(T_PLC_MS());

(* reset outputs, they should only be active 1 cycle *)
short := FALSE;
Middle := FALSE;
long := FALSE;

(* detect rising edge *)
IF in AND NOT edge THEN
	edge := TRUE;
	tn := tx;

(* detect for falling edge *)
ELSIF NOT in AND edge THEN
	edge := FALSE;
	tn := tx - tn;
	IF tn < t_short THEN
		short := TRUE;
	ELSIF tn > t_long THEN
		long := TRUE;
	ELSE
		Middle := TRUE;
	END_IF;

(* generate long pulse as soon as T_long is reached *)
ELSIF in AND tx - tn > t_long THEN
	long := TRUE;
END_IF;


(* revision history

hm	15. feb 2006	rev 1.0
	original version

hm	15 sep 2007		rev 1.1
	replaced Time() with T_PLC_MS for compatibility and performance reasons

*)
END_FUNCTION_BLOCK

(* POU Building/electrical/switch_I, ST *)
FUNCTION_BLOCK switch_I
VAR_INPUT
	set : BOOL;
	in : BOOL;
	rst : BOOL;
END_VAR
VAR_INPUT CONSTANT
	T_debounce : TIME := T#10ms;
	T_reconfig : TIME := T#1s;
	T_on_max : TIME := T#0h;
END_VAR
VAR_OUTPUT
	Q : BOOL := 0;
END_VAR
VAR
	state : BYTE := 0;
	edge : BOOL := 0;
	r_edge : BOOL := 0;
	T_on : TIME;
	tx: TIME;
END_VAR

(*
version 1.1	15 sep 2007
programmer 	oscat
tested by		tobias

this is an intelligent switch interface which has an autodetect feature for in and it will detect the type of switch connected automatically
the input can be connected to low active pulses, high active pulses and on/off switch.
it will automatically adjust to the correct type without manual adjustment
a configurable debounce timer will debounce input signals
if t_on_max is set to anything other then 0 the output will be turned off after the max on time is reached.

*)
(* read system time *)
tx := DWORD_TO_TIME(T_PLC_MS());

(* asynchronous set and reset first *)
IF set AND NOT rst THEN
	Q := 1;
	T_on := tx;
ELSIF rst THEN
	Q := 0;
(* check FOR input edge AND start debounce timer *)
ELSIF (in XOR edge) AND NOT (state = 1) THEN
	state := 1;
	T_on := Tx;
(* edge was detected and debounce time elapsed *)
ELSIF (state = 1) AND (Tx - t_debounce >= T_on) THEN
	state := 2;
	(* react on rising or falling edge depending on r_edge *)
	IF r_edge XOR in THEN Q := NOT Q; END_IF;
(* wait for T_reconfig and adjust r_edge *)
ELSIF state = 2 AND Tx - t_reconfig >= T_on THEN
	r_edge := in;
END_IF;
IF Q AND T_on_max > t#0ms AND Tx >= T_on + T_on_max THEN
	Q := FALSE;
END_IF;
edge := in;

(* revision history

hm	4 aug 2006	rev 1.0
	original version

hm	15.9.2007	rev 1.1
	replaced Time() with T_PLC_MS for compatibility and performance reasons

*)
END_FUNCTION_BLOCK

(* POU Building/electrical/Switch_X, ST *)
FUNCTION_BLOCK Switch_X
VAR_INPUT
	IN1 : BOOL;
	IN2 : BOOL;
	IN3 : BOOL;
	IN4 : BOOL;
	IN5 : BOOL;
	IN6 : BOOL;
END_VAR
VAR_OUTPUT
	Q1 : BOOL;
	Q2 : BOOL;
	Q3 : BOOL;
	Q4 : BOOL;
	Q5 : BOOL;
	Q6 : BOOL;
	Q31 : BOOL;
	Q41 : BOOL;
	Q51 : BOOL;
	Q61 : BOOL;
	Q32 : BOOL;
	Q42 : BOOL;
	Q52 : BOOL;
	Q62 : BOOL;
END_VAR
VAR_INPUT CONSTANT
	t_debounce : TIME := t#50ms;
END_VAR
VAR
	init : BOOL;
	T1, T2, T3, T4, T5, T6 : TOF;
	tx: TIME;
	x1: BOOL;
	x2: BOOL;
	E1, E2 : BOOL;
END_VAR

(*
version 1.0	15 Feb 2007
programmer 	oscat
tested by		tobias

*)
(* initialize on startup *)
IF NOT init THEN
	init := TRUE;
	IF t_debounce < t#50ms THEN tx := t#50ms; ELSE tx := t_debounce; END_IF;
	T1(PT := Tx);
	T2(PT := Tx);
	T3(PT := Tx);
	T4(PT := Tx);
	T5(PT := Tx);
	T6(PT := Tx);
ELSE
	Q1 := FALSE;
	Q2 := FALSE;
	Q3 := FALSE;
	Q4 := FALSE;
	Q5 := FALSE;
	Q6 := FALSE;
	Q31 := FALSE;
	Q41 := FALSE;
	Q51 := FALSE;
	Q61 := FALSE;
	Q32 := FALSE;
	Q42 := FALSE;
	Q52 := FALSE;
	Q62 := FALSE;
END_IF;

(* read inputs and debounce *)
	T1(IN := IN1);
	T2(IN := IN2);
	T3(IN := IN3);
	T4(IN := IN4);
	T5(IN := IN5);
	T6(IN := IN6);

(* detect edge of IN1 and IN2 *)
IF t1.Q AND NOT E1 THEN X1 := TRUE; END_IF;
IF t2.Q AND NOT E2 THEN X2 := TRUE; END_IF;

IF t1.Q THEN
	IF t3.q THEN
		q31 := TRUE;
		X1 := FALSE;
	ELSIF t4.q THEN
		q41 := TRUE;
		X1 := FALSE;
	ELSIF t5.q THEN
		q51 := TRUE;
		X1 := FALSE;
	ELSIF t6.q THEN
		q61 := TRUE;
		X1 := FALSE;
	END_IF;
ELSIF t2.Q THEN
	IF t3.q THEN
		q32 := TRUE;
		X2 := FALSE;
	ELSIF t4.q THEN
		q42 := TRUE;
		X2 := FALSE;
	ELSIF t5.q THEN
		q52 := TRUE;
		X2 := FALSE;
	ELSIF t6.q THEN
		q62 := TRUE;
		X2 := FALSE;
	END_IF;
(* in1 was active alone *)
ELSIF NOT T1.Q AND E1 AND X1 THEN
	Q1 := TRUE;
	X1 := FALSE;
ELSIF NOT T2.Q AND E2 AND X2 THEN
	Q2 := TRUE;
	X2 := FALSE;
ELSIF T3.Q THEN
	Q3 := TRUE;
ELSIF T4.Q THEN
	Q4 := TRUE;
ELSIF T5.Q THEN
	Q5 := TRUE;
ELSIF T6.Q THEN
	Q6 := TRUE;
END_IF;

(* save state of in1 and in2 *)
E1 := T1.Q;
E2 := T2.Q;
END_FUNCTION_BLOCK

(* POU Building/electrical/timer_1, ST *)
FUNCTION_BLOCK timer_1
VAR_INPUT
	DT_in : DT;
	start_time : TOD;
	duration : TIME;
	start_day : INT := 0;
END_VAR
VAR_OUTPUT
	Q : BOOL;
END_VAR
VAR
	last_check : TIME := T#0s;
	last: DATE := D#2041-01-01;
	dat: DATE;
	init : BOOL;
	tx: TIME;
	pulse_start: TIME;
END_VAR

(*
version 1.5	1. okt 2007
programmer 	oscat
tested by		tobias

this is a simple timer that generates an output pulse once a day if start_day = 0.
if start_day is a number from 1 .. 7 then a output pulse is generated for the respective weekday 1 = monday.
the output pulse width can be programmed, if set to 0 a pulse is generated for one cycle only.

*)
(* read system timer *)
tx := DWORD_TO_TIME(T_PLC_MS());

(* init on startup *)
IF NOT init THEN
	init := TRUE;
	last_check := tx - t#100ms;
END_IF;

(* check every 100ms *)
IF tx - last_check >= T#100ms THEN
	dat := DT_TO_DATE(dt_in);
	IF NOT Q AND (start_day = 0 OR start_day = weekday(dat)) AND dat <> last AND DT_TO_TOD(dt_in) >= start_time THEN
		Q := TRUE;
		last := dat;
		pulse_start := tx;
	ELSIF Q AND tx - pulse_start >= duration THEN
		Q := FALSE;
	END_IF;
	last_check := tx;
END_IF;

(*
1.12.2006 hm		rev 1.1
	corrected an error with pulse width = 0.

25.12.2006 hm	rev 1.2
	corrected an error when timer overflows.

14.apr 2007 hm	rev 1.3
	corrected an error while while output would not go active when start year would be 1970.
	increase accuracy by checking every 100ms
	added init section to compensate for timer overflow

15.9.2007	hm		rev 1.4
	replaced Time() with T_PLC_MS for compatibility and performance reasons

hm	1. okt 2007		rev 1.5
	corrected an error while output would not stay active over midnight.

*)
END_FUNCTION_BLOCK

(* POU Time&Date/weekday, ST *)
FUNCTION weekday : INT
VAR_INPUT
	idate : DATE;
END_VAR
VAR
END_VAR

(*
version 1.2	23 dec 2007
programmer 	hugo
tested by		tobias

calculates the weekday of a week according to ISO8601   
monday = 1 ..... sunday = 7  

*)
IF step7 THEN
	weekday := DWORD_TO_INT((DATE_TO_DWORD(idate)/86400+6) MOD 7) + 1;
ELSE
	weekday := DWORD_TO_INT((DATE_TO_DWORD(idate)/86400+3) MOD 7) + 1;
END_IF;
(* revision history
hm 21.8.06 rev 1.1
	corrected a miscalculation

hm	23.12.2007	rev 1.2
	correction for step7

*)
END_FUNCTION

(* POU Building/electrical/timer_2, ST *)
FUNCTION_BLOCK timer_2
VAR_INPUT
	DT_in : DT;
	start : TOD;
	duration : TIME;
	mode : BYTE;
	holiday : BOOL;
END_VAR
VAR_OUTPUT
	Q : BOOL;
END_VAR
VAR
	last_check : TIME := T#0s;
	dat : DATE;
	daytime : TOD;
	activation: TIME;
	tx: TIME;
	enabled: BOOL;
	wday: INT;
	init: BOOL;
END_VAR

VAR RETAIN
	run_date : DATE;
END_VAR

(*
version 1.2	15 sep 2007
programmer 	oscat
tested by		tobias

this timer generated programmabe output pulses per day, week, month and so on.
the mode input determines on which days the timer will be active.
	mode = 0			never
	mode = 1..7		monday .. sunday
	mode = 11			every day
	mode = 12			every second day
	mode = 13			every 3rd day
	mode = 14			every 4th day
	mode = 15			every 5th day
	mode = 16 		every 6th day
	mode = 20			only monday - friday
	mode = 21			only sat - sunday
	mode = 22			workdays only
	mode = 23			holidays and weekend
	mode = 24			holidays only
	mode = 25			every 1st day of the month
	mode = 26			every last day of the month
	mode = 27			every 31 of december
	mode = 28			every 1st of january

a holiday input can be used to supply holiday information to the module.
*)
(* read system time *)
tx := DWORD_TO_TIME(T_PLC_MS());

IF NOT init THEN
	init := TRUE;
	last_check := tx - t#100ms;
END_IF;

(* for performance resons exit if execution is not necessary *)
IF tx - last_check <= T#100ms THEN RETURN; END_IF;

(* calculate temp variables *)
dat := DT_TO_DATE(dt_in);
daytime := DT_TO_TOD(dt_in);
wday := weekday(dat);

(* calculate if any action is necessary today *)
enabled := FALSE;
CASE mode OF
1..7:	(* mondays to fridays *)
	IF wday = mode THEN enabled := 1; END_IF;
11:	(* every day *)
	enabled := TRUE;
12..16:	(* every nth day *)
	IF (TRUNC(DATE_TO_DWORD(dat)/86400)) MOD (mode - 10) = 0 THEN enabled := 1; END_IF;
20:	(* monday - friday *)
	IF wday <= 5 THEN enabled := TRUE; END_IF;
21:	(* saturday and sunday *)
	IF wday > 5 THEN enabled := TRUE; END_IF;
22: (* workdays only *)
	IF wday <= 5 AND NOT holiday THEN enabled := TRUE; END_IF;
23:	(* holidays and weekends *)
	IF wday > 5 OR holiday THEN enabled := TRUE; END_IF;
24:	(* holidays only *)
	enabled := holiday;
25:	(* 1st day of the month *)
	IF day_of_month(dat) = 1 THEN enabled := TRUE; END_IF;
26:	(* last day of month *)
	IF day_of_month(dat + t#1d) = 1 THEN enabled := TRUE; END_IF;
27:	(* 31st of december *)
	IF day_of_month(dat) = 31 AND month(dat) = 12 THEN enabled := TRUE; END_IF;
28:	(* 1st of january *)
	IF day_of_year(dat) = 1 THEN enabled := TRUE; END_IF;
END_CASE;

(* set or reset output if necessary *)
IF enabled AND NOT Q AND daytime >= start AND run_date <> dat THEN
	Q := 1;
	activation := tx;
	run_date := dat;
ELSIF Q AND tx - activation >= duration THEN
	Q := 0;
END_IF;
last_check := Tx;


(* revision history
hm 22.2.2007		rev 1.1
	changed VAR RETAIN PERSISTENT to VAR RETAIN for better compatibility
	wago lon contollers do not support persisitent

hm	15.9.2007		rev 1.2
	replaced Time() with T_PLC_MS for compatibility and performance reasons
 
*)
END_FUNCTION_BLOCK

(* POU Time&Date/holiday, ST *)
FUNCTION_BLOCK holiday
VAR_INPUT
	date_in : DATE;
END_VAR
VAR_INPUT CONSTANT
	size : INT := 24;
	feiertag : ARRAY [0..24] OF STRING(27) := 'Neujahr', 'Heilig Drei Könige', 'Karfreitag', 'Ostersonntag', 'Ostermontag', 'Tag der Arbeit',
	'Christi Himmelfahrt', 'Pfingstsonntag', 'Pfingstmontag', 'Fronleichnam', 'Augsburger Friedensfest', 'Maria Himmelfahrt',
	'Tag der Deutschen Einheit', 'Reformationstag', 'Allerheiligen', 'Buss und Bettag', '1. Weihnachtstag', '2. Weihnachtstag';
	f_day : ARRAY [0..24] OF SINT := 1, 6, -2, 0, 1, 1, 39, 49, 50 , 60, 8, 15, 3, 31, 1, 23, 25, 26;
	f_month : ARRAY [0..24] OF SINT := 1, 1, 0, 0, 0, 5, 0, 0, 0, 0, 8, 8, 10, 10, 11, 11, 12, 12;
	(* if month = 0 then F_day is the offset in days from easter *)
	f_use : ARRAY [0..24] OF SINT := 1,1,1,1,1,1,1,1,1,1,0,1,1,0,1,0,1,1;
	(* 0 = not used, 1 = used, -1..-7 menas the weekday before the specified date example -3 means wednesday before 23.11 *)
	Friday : BOOL := FALSE;
	Saturday : BOOL := FALSE;
	Sunday : BOOL := FALSE;
END_VAR
VAR_OUTPUT
	Y : BOOL;
	name : STRING(20);
END_VAR
VAR
	last_active : DATE;
	ostern: DATE;
	i: INT;
	jahr: INT;
	x_date: DATE;
	wday : INT;
END_VAR

(*
version 1.3	24 nov 2007
programmer 	hugo
tested by		tobias

holiday calculates if a given day is a holiday and displays the name of the holiday as string as well as a boolean flag to indicate a holiday.
the holidays can be specified in an array in the constants section of the function block.
a holiday can be of fixed date for example new years day on january 1st.
a holiday can have a fixed offset from easter sunday as for most church holidays.
a holiday can be a specific weekday before a fixed date, for example buss und bettag is the last wednesday before nov 23rd.
with a simple f_use flag any specific holiday can be turned on or off if needed.
The setup Variables Friday, Saturday and Sunday can be used to activate the output on the specific weekday.

*)
(* for performance reasons only activate once a day *)
IF last_active = date_in THEN RETURN; END_IF;

(* berechnung von ostern für das aktuelle jahr *)
jahr := year(date_in);
Ostern := easter(jahr);
last_active := Date_in;

(* check array if today is holiday *)
Y := FALSE;
name := '';
FOR i := 0 TO size DO
	x_date := set_Date(jahr, f_month[i], f_day[i]);
	IF f_use[i] = 1 AND f_month[i] > 0 THEN
		(* check for fixed date holiday *)
		IF x_date = date_in THEN
			Y := TRUE;
			name := feiertag[i];
			RETURN;
		END_IF;
	ELSIF f_use[i] = 1 AND f_month[i] = 0 THEN
		(* check for holiday in reference to easter *)
		IF date_add(ostern,f_day[i] ,0,0,0) = date_in THEN
			Y := TRUE;
			name := feiertag[i];
			RETURN;
		END_IF;
	ELSIF f_use[i] < 0 THEN
		(* check for holiday on a weekday before date *)
		IF weekday(date_in) = ABS(f_use[i]) AND date_in < x_date AND date_in >= date_add(x_date,-7,0,0,0) THEN
			Y := TRUE;
			name := feiertag[i];
			RETURN;
		END_IF;
	END_IF;
END_FOR;

wday := weekday(date_in);
IF wday = 7 AND Sunday THEN
	Y := TRUE;
ELSIF wday = 6 AND Saturday THEN
	Y := TRUE;
ELSIF wday = 5 AND Friday THEN
	Y := TRUE;
END_IF;

(* revision history
hm 27.2.2007		rev 1.1
	deleted unused variable init

hm	31 oct 2007	rev 1.2
	changed holiday definition from constant to input constant to allow easier changes by user without recompilation of the lib

hm 24 nov 2007	rev 1.3
	changes F_use of  Buß_und_Bettag to 0 because this is no official holiday
*)

(*
Neujahrstag 	1. Januar 	• 	• 	• 	• 	• 	• 	• 	• 	• 	• 	• 	• 	• 	• 	• 	•
Heilige Drei Könige 	6. Januar 	• 	• 												• 		
Karfreitag 	Ostersonntag - 2d 	• 	• 	• 	• 	• 	• 	• 	• 	• 	• 	• 	• 	• 	• 	• 	•
Ostersonntag 	siehe Osterdatum 				(•) 												
Ostermontag 	Ostersonntag + 1d 	• 	• 	• 	• 	• 	• 	• 	• 	• 	• 	• 	• 	• 	• 	• 	•
Tag der Arbeit 	1. Mai 	• 	• 	• 	• 	• 	• 	• 	• 	• 	• 	• 	• 	• 	• 	• 	•
Christi Himmelfahrt 	Ostersonntag + 39d 	• 	• 	• 	• 	• 	• 	• 	• 	• 	• 	• 	• 	• 	• 	• 	•
Pfingstsonntag 	Ostersonntag + 49d 				(•) 												
Pfingstmontag 	Ostersonntag + 50d 	• 	• 	• 	• 	• 	• 	• 	• 	• 	• 	• 	• 	• 	• 	• 	•
Fronleichnam 	Ostersonntag + 60d 	• 	• 					• 			• 	• 	• 	1) 			2)
Augsburger Friedensfest 	8. August 		(3) 														
Mariä Himmelfahrt 	15. August 		(5) 										• 				
Tag der Deutschen Einheit 	3. Oktober 6) 	• 	• 	• 	• 	• 	• 	• 	• 	• 	• 	• 	• 	• 	• 	• 	•
Reformationstag 	31. Oktober 				• 				• 					• 	• 		•
Allerheiligen 	1. November 	• 	• 								• 	• 	• 				
Buß- und Bettag 4) 	Mittwoch vor dem 23.11. 			7 										• 			
1. Weihnachtstag 	25. Dezember 	• 	• 	• 	• 	• 	• 	• 	• 	• 	• 	• 	• 	• 	• 	• 	•
2. Weihnachtstag 	26. Dezember 	• 	• 	• 	• 	• 	• 	• 	• 	• 	• 	• 	• 	• 	• 	• 	•
*)
END_FUNCTION_BLOCK

(* POU Time&Date/year, ST *)
FUNCTION year : INT
VAR_INPUT
	idate : DATE;
END_VAR
VAR
END_VAR

(*
version 1.2	23 dec 2007
programmer 	hugo
tested by		tobias

returs the year of a date  
the function works for dates from 1970 - 2099 

*)
IF Step7 THEN
	year := DWORD_TO_INT((DATE_TO_DWORD(idate)+43200) / 31557600 + 1990);
ELSE
	year := DWORD_TO_INT((DATE_TO_DWORD(idate)+43200) / 31557600 + 1970);
END_IF;

(* code used prior to rev 1.1
year := DWORD_TO_INT((DATE_TO_DWORD(idate)/864+71954300)/36525);
*)

(* revision history
hm	4. aug 2006		rev 1.0
	original version

hm	1. okt 2007		rev 1.1
	corrected error in algorithm
	adjustment for S7 compatibility

hm	23.12.2007		rev 1.2
	changed code for better performance
*)
END_FUNCTION

(* POU Time&Date/easter, ST *)
FUNCTION easter : DATE
VAR_INPUT
	year : INT;
END_VAR
VAR
	b,c: INT;
	oday: INT;
	omon: INT;
END_VAR

(*
version 1.1	15 dec 2007
programmer 	hugo
tested by		tobias

easter calculates the day of easter sunday for a given year.
most other catholic holidays are calculated in reference to easter sunday.

*)
(* this algorithms is 95 us *)

b := (204 - 11 * (year MOD 19)) MOD 30;
IF b = 28 OR b = 29 THEN b := b - 1; END_IF;
c := (year + SHR(year,2) + b - 13) MOD 7;
oday := 28 + b - c;
IF oday > 33 THEN
    oday := oday - 31;
    omon := 4;
ELSE
	omon := 3;
END_IF;

easter := set_Date(year, omon, oday);


(* this algorithm is 180 us
a := year MOD 19;
b := year / 100;
c := year MOD 100;
d := b / 4;
e := b MOD 4;
f := (b + 8) / 25;
g := (b - f + 1) / 3;
h := (19 * a + b - d -g + 15) MOD 30;
i := C / 4;
k := c MOD 4;
l := (32 + 2*e + 2*i - h - k) MOD 7;
m := (a + 11 * h + 22 * l) / 451;
x := h + l - 7 * m + 114;
n := X / 31;
o := x MOD 31 + 1;

easter := set_Date(year,n,o);
*)
(*
Im Magazin "Nature" vom 20. April 1876 veröffentlichte ein anonymer Autor eine Tabelle mit Regeln zur Berechnung des (Gregorianischen) Ostersonntages des Jahres J. In Formeln ausgedrückt erhält man das Folgende:
a	=	J mod 19
b	=	int(J / 100)
c	=	J mod 100
d	=	int(b / 4)
e	=	b mod 4
f	=	int((b + 8) / 25)
g	=	int((b - f + 1) / 3
h	=	(19 · a + b - d - g + 15) mod 30
i	=	int(c / 4)
k	=	c mod 4
l	=	(32 + 2 · e + 2 · i - h - k) mod 7
m	=	int((a + 11 · h + 22 · l) / 451)
n	=	int((h + l - 7 · m + 114) / 31)
o	=	(h + l - 7 · m + 114) mod 31

n ist hierbei die Nummer des Monats, o + 1 die Nummer des Tages auf welchen der Ostersonntag im Jahr J fällt. Dieser Algorithmus kommt ohne Hilfszahlen aus.

*)

(* revision history
hm	27. dec 2006	rev 1.0
	original version

hm	15. dec 2007	rev 1.1
	modified code for better performance

*)
END_FUNCTION

(* POU Time&Date/set_Date, ST *)
FUNCTION set_Date : DATE
VAR_INPUT
	year : INT;
	month : INT;
	day : INT;
END_VAR
VAR
	count : DWORD;
	leap: BOOL;
END_VAR

(*
version 1.2	1 okt 2007
programmer 	hugo
tested by		tobias

creates a date output from year, month and day of month   

*)
leap := leap_year(year);
IF STEP7 THEN
	count := SHR((year-1)*1461-2905932+day*4,2);
ELSE
	count := SHR((year-1)*1461-2876712+day*4,2);
END_IF;
(* old code before rev 1.3
leap := leap_year(year);
IF STEP7 THEN
	count := TRUNC((year-1)*365.25-726483+day);
ELSE
	count := TRUNC((year-1)*365.25-719178+day);
END_IF;
*)

CASE month OF
2:	count := count + 31;
3:	IF leap THEN count := count + 60; ELSE count := count + 59; END_IF;
4:	IF leap THEN count := count + 91; ELSE count := count + 90; END_IF;
5:	IF leap THEN count := count + 121; ELSE count := count + 120; END_IF;
6:	IF leap THEN count := count + 152; ELSE count := count + 151; END_IF;
7:	IF leap THEN count := count + 182; ELSE count := count + 181; END_IF;
8:	IF leap THEN count := count + 213; ELSE count := count + 212; END_IF;
9:	IF leap THEN count := count + 244; ELSE count := count + 243; END_IF;
10:	IF leap THEN count := count + 274; ELSE count := count + 273; END_IF;
11:	IF leap THEN count := count + 305; ELSE count := count + 304; END_IF;
12:	IF leap THEN count := count + 335; ELSE count := count + 334; END_IF;
END_CASE;
set_Date := DWORD_TO_DATE(count * 86400);


(* revision history
hm	4. aug. 2006	rev 1.0
	original version

hm	19 sep. 2007	rev 1.1
	use function leap_year to calculate leap year, more exceptions are handled

hm	1. okt	2007	rev 1.2
	added compatibility to step7

hm	16.dec 2007		rev 1.3
	changed code to improove performance
*)
END_FUNCTION

(* POU Time&Date/month, ST *)
FUNCTION month : INT
VAR_INPUT
	idate : DATE;
END_VAR
VAR
END_VAR

(*
version 1.1	1 okt 2007
programmer 	hugo
tested by		tobias

returns the month of a year

*)
month := day_of_year(idate);
IF leap_of_Date(idate) THEN
	CASE month OF
		1..31 	:	month := 1;
		32..60	:	month := 2;
		61..91	:	month := 3;
		92..121 :	month := 4;
		122..152:	month := 5;
		153..182:	month := 6;
		183..213:	month := 7;
		214..244:	month := 8;
		245..274:	month := 9;
		275..305:	month := 10;
		306..335:	month := 11;
		336..366:	month := 12;
	END_CASE;
ELSE
	CASE month OF
		1..31 	:	month := 1;
		32..59	:	month := 2;
		60..90	:	month := 3;
		91..120 :	month := 4;
		121..151:	month := 5;
		152..181:	month := 6;
		182..212:	month := 7;
		213..243:	month := 8;
		244..273:	month := 9;
		274..304:	month := 10;
		305..334:	month := 11;
		335..365:	month := 12;
	END_CASE;
END_IF;


(* old code used in rev 1.0
month := STRING_TO_INT(MID(DATE_TO_STRING(idate),2,8));
*)

(* revision history
hm	1. aug 2006		rev 1.0
	original version	

hm	1. okt 2007		rev 1.1
	replaced old code (string conversion) with mathematics
	the execution time is now multiple times faster.

*)
END_FUNCTION

(* POU Time&Date/day_of_year, ST *)
FUNCTION day_of_year : INT
VAR_INPUT
	idate : DATE;
END_VAR
VAR
END_VAR

(*
version 1.1	1 oct 2007
programmer 	hugo
tested by		tobias

calculates the day of the year 

*)
IF step7 THEN
	day_of_year := DWORD_TO_INT(DATE_TO_DWORD(idate)/86400 + 726483 - TRUNC((year(idate)-1)*365.25));
ELSE
	day_of_year := DWORD_TO_INT(DATE_TO_DWORD(idate)/86400 + 719178 - TRUNC((year(idate)-1)*365.25));
END_IF;

(* revivision history
hm	4. aug 2007		rev 1.0
	original version

hm	1. okt 2007		rev 1.1
	added compatibility to STEP7

*)
END_FUNCTION

(* POU Time&Date/leap_of_Date, ST *)
FUNCTION leap_of_Date : BOOL
VAR_INPUT
	idate : DATE;
END_VAR
VAR
END_VAR

(*
version 1.1	2 oct 2006
programmer 	hugo
tested by		tobias


leap_year is true if the tested year is a leap year  

*)
leap_of_Date := leap_year(year(idate));


(* change history

2.10.2006		changes to rev 1.1
the function now calls leap_year to accomodate further accuracy.
the function now works for any year from 1970 to 2100

*)
END_FUNCTION

(* POU Time&Date/leap_year, ST *)
FUNCTION leap_year : BOOL
VAR_INPUT
	yr : INT;
END_VAR
VAR
END_VAR

(*
version 1.1	2 oct 2006
programmer 	hugo
tested by		tobias


leap_year is true if the tested year is a leap year  
execution time on wago 750-841 =  12 us    
*)
leap_year := SHL(yr,14) = 0;

(* this code was used prior to rev 1.1

IF yr MOD 400 = 0 THEN leap_year := TRUE;
ELSIF yr MOD 100 = 0 THEN leap_year := FALSE;
ELSIF yr MOD 4 =0 THEN leap_year := TRUE;
ELSE leap_year := FALSE;
END_IF;

*)

(* change history

hm 	2.10.2006		rev 1.1
	the function now works for any year from 1970 up to 2100

hm	1. oct 2007		rev 1.2
	chaged code for higher performance
*)
END_FUNCTION

(* POU Time&Date/date_add, ST *)
FUNCTION date_add : DATE
VAR_INPUT
	idate : DATE;
	D : INT;
	W : INT;
	M : INT;
	Y : INT;
END_VAR
VAR
	mo: INT;
	yr : INT;
END_VAR


(*
version 1.2	1 nov 2007
programmer 	hugo
tested by		tobias

date_add adds days, weeks, month or years to a date.
negative inputs are allowed for subtraction.

*)
date_add := DWORD_TO_DATE(DATE_TO_DWORD(idate) + 86400 * INT_TO_DWORD(d) + 604800 * INT_TO_DWORD(w));
yr := year(date_add) + y;
IF m > 0 THEN
	mo := month(date_add) + m;
	yr := yr + (mo - 1) / 12;
	mo := mo MOD 12;
	IF mo = 0 THEN mo := 12; END_IF;
	date_add := set_Date(yr, mo, day_of_month(date_add));
ELSIF m < 0 THEN
	mo := month(date_add) + m;
	yr := yr + mo / 12 -1;
	mo := mo MOD 12 + 12;
	date_add := set_Date(yr, mo, day_of_month(date_add));
ELSE
	date_add := set_Date(yr, month(date_add), day_of_month(date_add));
END_IF;

(* revision history

hm 27.12.2006	rev 1.0

hm 12.4.2007		rev 1.1
	corrected an error while date would be incorrect when year  = 0

hm	1.11.2007		rev 1.2
	added int_to_dword stetements to avoid possible overrun with möller ecp4
*)
END_FUNCTION

(* POU Time&Date/day_of_month, ST *)
FUNCTION day_of_month : INT
VAR_INPUT
	idate : DATE;
END_VAR
VAR
	yd: INT;
END_VAR

(*
version 1.3	8. okt 2007
programmer 	hugo
tested by		tobias

returns the day OF month for any DATE

*)
yd := day_of_year(idate);
IF leap_of_Date(idate) THEN
	CASE yd OF
		1..31 	:	day_of_month := yd;
		32..60	:	day_of_month := yd - 31;
		61..91	:	day_of_month := yd - 60;
		92..121 :	day_of_month := yd - 91;
		122..152:	day_of_month := yd - 121;
		153..182:	day_of_month := yd - 152;
		183..213:	day_of_month := yd - 182;
		214..244:	day_of_month := yd - 213;
		245..274:	day_of_month := yd - 244;
		275..305:	day_of_month := yd - 274;
		306..335:	day_of_month := yd - 305;
		336..366:	day_of_month := yd - 335;
	END_CASE;
ELSE
	CASE yd OF
		1..31 	:	day_of_month := yd;
		32..59	:	day_of_month := yd - 31;
		60..90	:	day_of_month := yd - 59;
		91..120 :	day_of_month := yd - 90;
		121..151:	day_of_month := yd - 120;
		152..181:	day_of_month := yd - 151;
		182..212:	day_of_month := yd - 181;
		213..243:	day_of_month := yd - 212;
		244..273:	day_of_month := yd - 243;
		274..304:	day_of_month := yd - 273;
		305..334:	day_of_month := yd - 304;
		335..365:	day_of_month := yd - 334;
	END_CASE;
END_IF;


(*
this function is simple but took too long with 133 us
the problem is date_to_string is far too slow
day_of_month := STRING_TO_INT(RIGHT(DATE_TO_STRING(idate),2));

Revision history

hm 22.1.2007		rev 1.1
	deleted unused variable day_in_year and day_in_year_begin

hm	1. okt 2007		rev 1.2
	changed code to use day_of_year and leap_of_date
	added compatibility to STEP7

hm	8. oct 2007		rev 1.3
	deleted unused variable yr
*)
END_FUNCTION

(* POU Building/HLK/Air_density, ST *)
FUNCTION Air_density : REAL
VAR_INPUT
	T : REAL;
	P : REAL;
	RH : REAL;
END_VAR
VAR CONSTANT
	RL : REAL := 287.05;
	RX : REAL := 3.773319E-3;
END_VAR
VAR
END_VAR

(*
version 1.1	4 dec 2007
programmer 	hugo
tested by		tobias

this function calculates the air density between 0 and 100 deg C

*)
Air_density := PN * (1 - RH * SDD(T, TRUE) * RX / P) / (RL * ( T - TK));

(* original code used for rev 1.0

SDD := SDD(T,FALSE);
RF := RL / (1- RH*SDD/P*RX);
Air_density := P / (RF * (T-TK));

*)

(* revision history

hm	29.10.2007		rev 1.0
	original version

hm	4.12.2007		rev 1.1
	changed code for better performance

*)
END_FUNCTION

(* POU Building/HLK/SDD, ST *)
FUNCTION SDD : REAL
VAR_INPUT
	T : REAL;
	ICE: BOOL;
END_VAR
VAR CONSTANT
END_VAR
VAR
END_VAR

(*
version 1.1	2 dec 2007
programmer 	hugo
tested by		tobias

this function calculates the vapor saturation pressure for moist Air over ice or water

*)
IF ice THEN
	SDD := 611.153 * EXP(22.4433 * T / (272.186 + T));
ELSE
	SDD := 611.213 * EXP(17.5043 * T / (241.2 + T));
END_IF;

(* old code used in rev 1.0
IF ice THEN
	SDD := 611.153 * exp10(9.747*T / (272.186 + T));
ELSE
	SDD := 611.213 * exp10(7.602*T / (241.2 + T));
END_IF;
*)


(* revision history

hm 29 oct 2007		rev 1.0
	original version

hm	2. dec 2007		rev 1.1
	changed code for better performance
*)
END_FUNCTION

(* POU Building/HLK/Air_enthalpy, ST *)
FUNCTION Air_enthalpy : REAL
VAR_INPUT
	T : REAL;
	RH : REAL;
END_VAR
VAR CONSTANT
	CPL : REAL := 1.00482;
	CW : REAL := 1.86;
	LH : REAL := 2500.78;
END_VAR
VAR
END_VAR

(*
version 1.1	2 nov 2007
programmer 	hugo
tested by		tobias

this function calculates the enthalpy for humid air between 0 and 100 deg C

*)
Air_enthalpy := CPL * T + (CW * T + LH) * dew_con(RH,T);

(* revision history

hm	31.10.2007		rev 1.0
	original version

hm	2.11.2007		rev 1.1
	deleted unused variable RF

hm	2.12.2007		rev 1.2
	changed code for better performance
*)
END_FUNCTION

(* POU Building/HLK/dew_con, ST *)
FUNCTION dew_con : REAL
VAR_INPUT
	RH : REAL;
	T : REAL;
END_VAR
VAR CONSTANT
END_VAR
VAR
END_VAR

(*
version 1.2	2 dec 2007
programmer 	hugo
tested by		tobias

this function calculates the water concentratin in air for a given temperature and relative humidity.
the output states the concentration of water vapor in air in Gramms / qubic meter.

*)
IF rh > 0 THEN
(*	this code is good to read but need to be improoved
	SDD := 6.1078*EXPT(10,(a*T)/(b+T));
	DD := RH/100 * SDD;
	V := LOG(DD/6.1078);
	TD := b*V/(a-v);
	dew_con := 0.1 * mw / RU * DD / (T - TK);
*)
	dew_con := 2.166824303E-2 * RH * SDD(T,FALSE)  / (T - TK);
ELSE
	dew_con := 0;
END_IF;

(*
Bezeichnungen:
r = relative Luftfeuchte
T = Temperatur in °C
TK = Temperatur in Kelvin (TK = T + 273.15)
TD = Taupunkttemperatur in °C
DD = Dampfdruck in hPa
SDD = Sättigungsdampfdruck in hPa

Parameter:
a = 7.5, b = 237.3 für T >= 0
a = 7.6, b = 240.7 für T < 0 über Wasser (Taupunkt)
a = 9.5, b = 265.5 für T < 0 über Eis (Frostpunkt)

R* = 8314.3 J/(kmol*K) (universelle Gaskonstante)
mw = 18.016 kg (Molekulargewicht des Wasserdampfes)
AF = absolute Feuchte in g Wasserdampf pro m3 Luft

Formeln:

   1. SDD(T) = 6.1078 * 10^((a*T)/(b+T))
   2. DD(r,T) = r/100 * SDD(T)
   3. r(T,TD) = 100 * SDD(TD) / SDD(T)
   4. TD(r,T) = b*v/(a-v) mit v(r,T) = log10(DD(r,T)/6.1078)
   5. AF(r,TK) = 10^5 * mw/R* * DD(r,T)/TK; AF(TD,TK) = 10^5 * mw/R* * SDD(TD)/TK 

*)

(* revision history

hm 29 apr 2007		rev 1.0
	original version

hm	13.sep 2007		rev 1.1
	improoved coding for speed
	deleted unused variabled SDD,DD,V, TD

hm	2. dec 2007		rev 1.2
	changed code for better performance
	output is now in Gramms / Qubic meter
*)
END_FUNCTION

(* POU Building/HLK/Boiler, ST *)
FUNCTION_BLOCK Boiler
VAR_INPUT
	T_upper : REAL;
	T_lower : REAL;
	Pressure : BOOL := TRUE;
	enable : BOOL := TRUE;
	Req_1 : BOOL;
	Req_2 : BOOL;
	Boost : BOOL;
END_VAR
VAR_INPUT CONSTANT
	t_upper_min : REAL := 50;
	t_upper_max : REAL := 60;
	T_lower_enable : BOOL;
	T_lower_max : REAL := 60;
	T_request_1 : REAL := 70;
	T_request_2 : REAL := 50;
	T_request_hys : REAL := 5;
	T_protect_high : REAL := 80;
	T_protect_low : REAL := 10;
END_VAR
VAR_OUTPUT
	Heat : BOOL;
	error : BOOL;
	status : BYTE;
END_VAR
VAR
	edge: BOOL;
	boost_mode: BOOL;
	flag_0 : BOOL;
	flag_1: BOOL;
	flag_2: BOOL;
END_VAR

(*
version 1.0	27 feb 2007
programmer 	hugo
tested by		tobias

this function block controls a hot water boiler. The Boiler can be equipped with two temperature sensors on top and bottom of the tank, T_LOWER_ENABLE must be set to True in this case.
alternatively can BOILER be configured for one (TOP) temperature sensor only (T_LOWER_ENABLE set to False).
A Pressure sensor is used to detect fresh water pressure and disable all heating if there is no water pressure. This input is dset to True by default, so if it is not used it can simply be left open.
A enable input enables the hot water heating while it is set to True. alternatively can a Ture on Req_1 or Req_2 start the heating to predefined temperatures during setup.
A low to high edge on the boost input will start heating imediately until T_upper_max is reached, it can be used to generate extra hot water when needed.

*)
(* read sensors and check for valid data *)
IF t_upper > t_protect_high THEN
	status := 1;
	heat := FALSE;
	error := TRUE;
ELSIF t_upper < t_protect_low THEN
	status := 2;
	heat := TRUE;
	error := TRUE;
ELSIF t_lower > T_protect_high AND t_lower_enable THEN
	status := 3;
	heat := FALSE;
	error := TRUE;
ELSIF t_lower < t_protect_low AND t_lower_enable THEN
	status := 4;
	heat := TRUE;
	error := TRUE;
ELSIF NOT pressure THEN
	status := 5;
	heat := FALSE;
	error := TRUE;
ELSIF req_1 OR req_2 OR enable OR boost THEN
	error := FALSE;

	(* determine if heat needs to be turned on *)
	IF boost AND NOT edge AND t_upper < t_upper_max THEN
		status := 101;
		heat := TRUE;
		boost_mode := TRUE;
	ELSIF enable AND t_upper < T_upper_min THEN
		status := 102;
		heat := TRUE;
	ELSIF req_1 AND t_upper < T_request_1 THEN
		status := 103;
		heat := TRUE;
	ELSIF req_2 AND t_upper < t_request_2 THEN
		status := 104;
		heat := TRUE;
	END_IF;

	(* determine the shut off temperature *)
	IF heat THEN
		IF (enable OR boost_mode) THEN
			flag_0 := TRUE;
			IF T_lower_enable AND T_lower > T_lower_max THEN
				flag_0 := FALSE;
				boost_mode := FALSE;
			ELSIF NOT T_lower_enable AND T_upper > T_upper_max THEN
				flag_0 := FALSE;
				boost_mode := FALSE;
			END_IF;
		ELSE
			flag_0 := FALSE;
		END_IF;
		IF req_1 AND T_upper > T_request_1 + T_request_hys THEN flag_1 := FALSE; ELSE flag_1 := req_1; END_IF;
		IF req_2 AND T_upper > T_request_2 + T_request_hys THEN flag_2 := FALSE; ELSE flag_2 := req_2; END_IF;

		(* shut off heat if no longer needed *)
		heat := flag_0 OR flag_1 OR flag_2;
		IF heat = FALSE THEN status := 100; END_IF;
	END_IF;
ELSE
	status := 100;
	heat := FALSE;
	error := FALSE;
END_IF;
edge := boost;
END_FUNCTION_BLOCK

(* POU engineering/conversion/pressure, ST *)
FUNCTION_BLOCK pressure
VAR_INPUT
	mws : REAL;
	torr : REAL;
	att : REAL;
	atm : REAL;
	pa : REAL;
	bar : REAL;
END_VAR
VAR_OUTPUT
	Ymws : REAL;
	Ytorr : REAL;
	Yatt : REAL;
	Yatm : REAL;
	Ypa : REAL;
	Ybar : REAL;
END_VAR
VAR
END_VAR

(*
version 1.0	27 mar 2007
programmer 	hugo
tested by		oscat

this function converts different pressure units
any unused input can simply be left open.
different inputs connected at the same time will be added up.
*)
Ybar := bar +
		pa / 100000 +
		0.980665 * att +
		1.01325 * atm +
		0.001333224 * torr +
		0.0980665 * mws;
Ymws := ybar / 0.0980665;
Ytorr := ybar / 0.001333224;
Yatt := ybar / 0.980665;
yatm := ybar / 1.01325;
Ypa := ybar * 100000;


(*
Druck, Pascal Pa 1 Pa = 1 N/m2 = 1 kg/(s2 �E m) . 0,75 �E 10.2 mmHg
mechanische 1 MPa = 1 N/mm2 . fur Festigkeitsangaben
Spannung Bar bar 1 bar = 105 Pa = 103 mbar = 105 kg/(s2 �E m)
Millimeter- mmHg 1 mmHg = 133,322 Pa = 1,333 22 mbar
Quecksilbersaule . nur in Heilkunde zulassig
physik. Atmosphare atm 1 atm = 1,013 25 bar
techn. Atmosphare at 1 at = 1 kp/cm2 = 0,980665 bar
Torr Torr 1 Torr = (101325/760) Pa = 1,333224 mbar
Meter-Wassersaule mWS 1 mWS = 9806,65 Pa = 98,0665 mbar
psi lbf/in2 1 lbf/in2 = 68,947 57 mbar = 6894,757 Pa

*)
END_FUNCTION_BLOCK

(* POU Building/HLK/Burner, ST *)
FUNCTION_BLOCK Burner
VAR_INPUT
	in : BOOL;
	stage2 : BOOL;
	over_temp : BOOL;
	oil_temp : BOOL := TRUE;
	Flame : BOOL;
	rst : BOOL;
	rst_timer : BOOL;
END_VAR
VAR_INPUT CONSTANT
	pre_heat_time : TIME := t#5s;
	pre_vent_time : TIME := t#15s;
	pre_ignite_time : TIME := t#5s;
	post_ignite_time : TIME := t#25s;
	stage2_delay : TIME := t#10s;
	safety_time : TIME := t#5s;
	lockout_time : TIME := t#10s;
	multiple_ignition : BOOL := TRUE;
	KW1 : REAL;
	KW2 : REAL;
END_VAR
VAR_OUTPUT
	motor : BOOL;
	coil1 : BOOL;
	coil2 : BOOL;
	pre_heat: BOOL;
	ignite : BOOL;
	runtime1 : REAL;
	runtime2 : REAL;
	KWh : REAL;
	cycles : REAL;
	status : BYTE;
	fail : BOOL;
END_VAR
VAR
	state : BYTE;
	last : TIME;
	tx: TIME;
	last_change: TIME;
	timer1 : ontime;
	timer2 : ontime;
	oil_temp_last: BOOL;
END_VAR

(*
version 1.5	15 sep 2007
programmer 	oscat
tested by		tobias

burner ist eine Oel-Brenner_steuerung fuer nichtmodulierende Oelbrenner
die steuerung kann ueber setup werte programmiert werden und entsprechenden brennern angepasst werden.
die vorheizzeit ist die zeit die eine oelvorwaermung aufgeheizt wird bevor der motor gestartet wird.
der eingang oil_temp gibt an ob die oil_temp erreicht wurde, er ist default auf true und kann auch offen gelassen werden.
die vorbelueftungszeit ist die zeit die der luefter laeuft bevor die oelzufuhr freigegeben wird.
die vorzuendzeit iust diejenige zeit die die zuendung vor offnen des oelventiel gestartet wird.
nachzuendzeit ist die zeit die nach entzuendung der flamme noch gezuendet wird.
die sicherheitszeit ist die zeit nach der die oelzufuhr gesperrt wird wenn keine flamme entsteht.
nach ablauf der sicherheitszeit wird ein fehler flag gesetzt und kann erst nach der sperrzeit wieder durch einen reset geloescht werden.
waehrend der sperrzeit ist keine weitere zuendung oder einschalten moeglich.
das flag mehrfachzuendung gibt an ob eine erloschene flamme in betrieb automatisch wieder gezuendet werden soll.
der flammwaechster liegt auf eingang flamme, ein uebertemperaturschutz auf dem eingang over_temp
der betriebsstundenzaehler gibt die brennerstunden in stunden als real ausgabewer an.
der ausgang motor steuert den luefter / pumpenmotor, oil_ventil schaltet das oil ventil und zuendung schaltet die zuendung ein.

if output fail > 0 an error happened and the output has an error code:
0 :	no error
1 :	pre heating time expired and oil temp input is not true
2 :	flame monitor is active during preheating time
3 :	flame monitor active during pre_ventilation_time
4 :	no ignoition during safety time
5 :	no flame during operation
9 :	overtemp input is true

*)
(* read system time *)
tx := DWORD_TO_TIME(T_PLC_MS());

(* check rst input and overtemp *)
IF rst OR over_temp OR state = 0 THEN
	IF status > 0 AND tx - last_change >= lockout_time AND rst THEN
		status := 110;
		fail := FALSE;
		state := 1;
	ELSE
		(* normaler reset *)
		motor := FALSE;
		coil1 := FALSE;
		coil2 := FALSE;
		ignite := FALSE;
		pre_heat := FALSE;
		IF over_temp THEN
			status := 9;
			fail := TRUE;
		END_IF;
		last_change := tx;
		last := tx;
		state := 1;
	END_IF;
END_IF;

(* check for timer rst and rst timer if true *)
IF rst_timer THEN
	timer1( rst := TRUE);
	timer1.rst := FALSE;
	timer2(rst := TRUE);
	timer2.rst := FALSE;
END_IF;

(* quit here if an error is present *)
IF (status > 0 AND status < 100) OR rst THEN RETURN; END_IF;

(* start sequence *)
CASE state OF

1:	(* in signal starts oil pre heating *)
	IF in AND flame THEN
		state := 7;
		pre_heat := FALSE;
		status := 2;
		last_change := tx;
	ELSIF in THEN
		pre_heat := TRUE;
		state := 2;
		last_change := tx;
	END_IF;

2:	(* after pre_heating time start motor *)
	IF (tx- last_change >= pre_heat_time AND oil_temp) OR (oil_temp AND NOT oil_temp_last) THEN
		motor := TRUE;
		state := 3;
		last_change := tx;
	(* pre_heat_time ist abgelaufen und oil_temp ist nicht aktiv *)
	ELSIF tx - last_change >= pre_heat_time AND NOT oil_temp THEN
		state := 7;
		pre_heat := FALSE;
		status := 1;
		last_change := tx;
	(* flame monitor cannot be active at this time *)
	ELSIF flame THEN
		state := 7;
		pre_heat := FALSE;
		status := 2;
		last_change := tx;
	END_IF;

3:	(* abwarten bis zündung eingeschaltet werden kann *)
	IF tx - last_change >= pre_vent_time - pre_ignite_time THEN
		ignite := TRUE;
		state := 4;
		last_change := tx;
	(* flame monitor cannot be active at this time *)
	ELSIF flame THEN
		state := 7;
		pre_heat := FALSE;
		motor := FALSE;
		status := 3;
		last_change := tx;
	END_IF;

4:	(* warten bis oelzufuhr geoeffnet werden darf *)
	IF tx - last_change >= pre_ignite_time THEN
		coil1 := TRUE;
		state := 5;
		last_change := tx;
	END_IF;

5:	(* warten auf flammwaechter und falls noetig abschalten *)
	IF tx - last_change >= safety_time OR flame THEN
		IF NOT flame THEN
			(* notabschaltung da flammwaechster nicht angesprochen hat *)
			state := 7;
			motor := FALSE;
			coil1 := FALSE;
			pre_heat := FALSE;
			ignite := FALSE;
			status := 4;
			last_change := tx;
		ELSE
			state := 6;
			last_change := tx;
		END_IF;
	END_IF;

6:	(* brenner läuft, flammueberwachung und nach ablauf der nachigniteszeit ignite abschalten *)
	IF NOT flame AND NOT multiple_ignition THEN
		(* notabschaltung da flammwaechster keine flamme meldet *)
		state := 7;
		motor := FALSE;
		coil1 := FALSE;
		coil2 := FALSE;
		pre_heat := FALSE;
		ignite := FALSE;
		status := 5;
		last_change := tx;
	ELSIF NOT flame AND multiple_ignition THEN
		ignite := TRUE;
		state := 5;
		coil2 := FALSE;
		last_change := tx;
	ELSE
		IF tx - last_change >= post_ignite_time THEN
			(* post_ignite_time abgelaufen, ignite abschalten *)
			ignite := FALSE;
		END_IF;
		IF tx - last_change >= stage2_delay AND stage2 THEN
			coil2 := TRUE;
		ELSE
			coil2 := FALSE;
		END_IF;
	END_IF;
END_CASE;

(* abschaltung wenn kein eingangssignal *)
IF NOT in THEN
	state := 1;
	motor := FALSE;
	coil1 := FALSE;
	coil2 := FALSE;
	ignite := FALSE;
	pre_heat := FALSE;
	last_change := tx;
END_IF;

(* runtimezähler *)
timer1(in := flame AND in AND motor AND coil1 AND NOT coil2);
timer2(in := flame AND in AND motor AND coil1 AND coil2);
runtime1 := timer1.ontime;
runtime2 := timer2.ontime;
cycles := timer1.cycles;
KWH := runtime1 * KW1 + runtime2 * KW2;

(* zeit fuer naechsten aufruf merken *)
last := tx;

(* set fail output IF ERROR and Status  if normal operation *)

IF status > 0 AND status < 100 THEN
	fail := TRUE;
ELSE
	fail := FALSE;
	IF NOT in THEN
		status := 110;
	ELSIF flame AND in AND motor AND coil2 AND coil1 THEN
		status := 113;
	ELSIF flame AND in AND motor AND coil1 THEN
		status := 112;
	ELSE
		status := 111;
	END_IF;
END_IF;


(*
31.12.2006	hm		rev 1.1
	added pre_heat timing and output
	flame monitor before ignition will generate error on status output
	added output for KWh

31.12.2006	hm		rev 1.2
	added oil_temp_input

31.12.2006	hm		rev 1.3
	changed status output to be byte instead of bool

22.1.2007		hm		rev 1.4
	renamed fail output to status
	added output cycles
	corrected an error while pre_heat would be on when an error was present
	added coil2 output and stage2 input

15.9.2007		hm		rev 1.5
	replaced Time() with T_PLC_MS for compatibility and performance reasons

*)
END_FUNCTION_BLOCK

(* POU Building/HLK/dew_rh, ST *)
FUNCTION dew_rh : REAL
VAR_INPUT
	VC : REAL;
	T : REAL;
END_VAR

(*
version 1.1	2 dec 2007
programmer 	hugo
tested by		tobias

this function calculates the relative humidity in air for a given temperature in °C and vapor concentration in Kg/m³..

*)
dew_rh := LIMIT(0,VC / dew_con(1,T),100);

(* code before rev 1.1
dew_rh := VC / dew_con(100,T) * 100;
IF dew_rh > 100 THEN dew_rh := 100; END_IF;
*)

(* revision history
hm		29. apr 2007	rev 1.0
	original version

hm		2. 12. 2007		rev 1.1
	new code for better performance

*)
END_FUNCTION

(* POU Building/HLK/dew_temp, ST *)
FUNCTION dew_temp : REAL
VAR_INPUT
	RH : REAL;
	T : REAL;
END_VAR
VAR CONSTANT
	a : REAL := 7.5;
	b : REAL := 237.3;
END_VAR
VAR
	V : REAL;
END_VAR

(*
version 1.3	2 dec 2007
programmer 	hugo
tested by		tobias

this function calculates the dew point for air given the temperature and relative humidity.
dew_temp(60,0.25) = 16.7 °C.
which means the dew point for air with 25° and 60% RH is at 16.7 °C.


*)
IF rh > 0 THEN
(*	old code was rewritten for better performance
	SDD := 6.1078*EXPT(10,(a*T)/(b+T));
	DD := RH/100 * SDD;
	V := LOG(DD/6.1078);
	dew_temp := b*V/(a-v);
*)
	V := LOG(RH/100 * exp10((a*T)/(b+T)));
	dew_temp := b*V/(a-V);
ELSE
	dew_temp:= -TK;
END_IF;

(* revision history

hm		2.10.2006	rev 1.0
	original version created

hm		29.4.2007	rev 1.1
	checked for rh not to be 0 because log(0) is not defined

hm		13.9.2007	rev 1.2
	code rewritten for better performance

hm		2. dec 2007	rev 1.3
	changed code for better performance
*)

(*
Bezeichnungen:
r = relative Luftfeuchte
T = Temperatur in °C
TK = Temperatur in Kelvin (TK = T + 273.15)
TD = Taupunkttemperatur in °C
DD = Dampfdruck in hPa
SDD = Sättigungsdampfdruck in hPa

Parameter:
a = 7.5, b = 237.3 für T >= 0
a = 7.6, b = 240.7 für T < 0 über Wasser (Taupunkt)
a = 9.5, b = 265.5 für T < 0 über Eis (Frostpunkt)

R* = 8314.3 J/(kmol*K) (universelle Gaskonstante)
mw = 18.016 kg (Molekulargewicht des Wasserdampfes)
AF = absolute Feuchte in g Wasserdampf pro m3 Luft

Formeln:

   1. SDD(T) = 6.1078 * 10^((a*T)/(b+T))
   2. DD(r,T) = r/100 * SDD(T)
   3. r(T,TD) = 100 * SDD(TD) / SDD(T)
   4. TD(r,T) = b*v/(a-v) mit v(r,T) = log10(DD(r,T)/6.1078)
   5. AF(r,TK) = 10^5 * mw/R* * DD(r,T)/TK; AF(TD,TK) = 10^5 * mw/R* * SDD(TD)/TK 

*)
END_FUNCTION

(* POU mathematical/exp10, ST *)
FUNCTION exp10 : REAL
VAR_INPUT
	X : REAL;
END_VAR
VAR
END_VAR

(*
version 1.0	 2 dec 2007
programmer 	hugo
tested by		tobias

this function calculates the exponent to the basis 10
exp10(3) = 1000

*)
exp10 := EXP(X * 2.30258509299405);

(* revision history
hm	2. dec 2007		rev 1.0
	original version

*)
END_FUNCTION

(* POU Building/HLK/Heat_index, ST *)
FUNCTION Heat_index : REAL
VAR_INPUT
	T : REAL;
	RH : REAL;
END_VAR
VAR
	RH2 : REAL;
	T2 : REAL;
END_VAR

(*
version 1.2	2 dec 2007
programmer 	hugo
tested by		tobias

this function calculates the heat index temperature depending on external temperature and Relative humidity

*)
IF RH < 20 OR T < 20 THEN
	Heat_index := T;
ELSE
	RH2 := RH * RH;
	T := C_to_F(T);
	T2 := T * T;
	Heat_index := -42.379 + 2.04901523 * T - 6.83783E-3 * T2
			+ RH * (10.1433127 - 0.22475541 * T + 1.22874E-3 * T2)
			+ RH2 * (8.5282E-4 * T - 5.481717E-2 - 1.99E-6 * T2);
	Heat_index := F_to_C(Heat_index);
END_IF;

(* revision history

hm 27.2.2007		rev 1.1
	deleted unused variables rh3 and T3

hm	2.12.2007		rev 1.2
	changed code for better performance
*)
END_FUNCTION

(* POU engineering/conversion/C_to_F, ST *)
FUNCTION C_to_F : REAL
VAR_INPUT
	celsius : REAL;
END_VAR
VAR
END_VAR

(*
version 1.0	4 aug 2006
programmer 	hugo
tested by		tobias

this function converts celsius  to fahrenheit 

*)
C_to_F := celsius * 1.8 + 32;
END_FUNCTION

(* POU engineering/conversion/F_to_C, ST *)
FUNCTION F_to_C : REAL
VAR_INPUT
	fahrenheit : REAL;
END_VAR
VAR
END_VAR

(*
version 1.0	4 aug 2006
programmer 	hugo
tested BY		tobias

this FUNCTION converts fahrenheit TO celsius

executioin TIME on wago 750-841 = 15us
*)
F_to_C := (fahrenheit -32) / 1.8;
END_FUNCTION

(* POU Building/HLK/heat_meter, ST *)
FUNCTION_BLOCK heat_meter
VAR_INPUT
	TF, TR : REAL;
	LPH : REAL;
	E : BOOL;
	RST : BOOL;
END_VAR
VAR_INPUT CONSTANT
	CP : REAL;
	Density : REAL;
	Content : REAL;
	Pulse_Mode : BOOL;
	Return_meter : BOOL;
	AVG_time : TIME := T#5s;
END_VAR
VAR_OUTPUT
	Y : REAL;
	C : REAL;
END_VAR
VAR
	tx, last : DWORD;
	int1 : FT_INT;
	edge : BOOL;
	X: REAL;
	init: BOOL;
	Y_last: REAL;
END_VAR

(*
version 1.1	25 dec 2007
programmer 	hugo
tested by		tobias

Heat meter measures the heat transfer of water of a mixture of water and another component.
The inputs are foreward temperature and reverse temperature.
the additional component is specified with its parameters density, Specific heat capacity and content in %.
an input e anables the measurement while it can be configured to be based on X liters / pulse or in liters / hour.
the output is in Joule.

*)
IF rst THEN
	int1(rst := TRUE);
	int1.rst := FALSE;
	C := 0;
	Y := 0;
ELSIF pulse_mode AND e AND NOT edge THEN
	IF return_meter THEN
		X := (Water_density(TR, FALSE) * (water_enthalpy(TF) - water_enthalpy(TR)) * (1-content) + CP * Density * content*(TF-TR));
	ELSE
		X := (Water_density(TF, FALSE) * (water_enthalpy(TF) - water_enthalpy(TR)) * (1-content) + CP * Density * content*(TF-TR));
	END_IF;
	Y := Y + X * LPH;
	edge := e;
ELSIF NOT pulse_mode AND e THEN
	IF return_meter THEN
		X := (Water_density(TR, FALSE) * (water_enthalpy(TF) - water_enthalpy(TR)) * (1-content) + CP * Density * content*(TF-TR));
	ELSE
		X := (Water_density(TF, FALSE) * (water_enthalpy(TF) - water_enthalpy(TR)) * (1-content) + CP * Density * content*(TF-TR));
	END_IF;
	int1(in := X * LPH / 3600.0, out_min := 0, out_max := 3E38);
	Y := int1.Out;
END_IF;

(* read system_time *)
tx := T_PLC_MS();

(* only init at startup necessary *)
IF NOT init THEN
	init := TRUE;
	last := tx;
END_IF;

(* calculate the current consumption *)
IF (tx - last >= TIME_TO_DWORD(AVG_TIME)) AND (avg_time > T#0s) THEN
	last := tx;
	C := (Y - Y_last) * 3.6/TIME_TO_DWORD(AVG_TIME);
	Y_last := Y;
END_IF;



(* revision history
hm		16.11.2007	rev 1.0
	original version

hm		24.12.2007	rev 1.1
	added config variable return_meter
	added output C for current consumption
*)
END_FUNCTION_BLOCK

(* POU Building/HLK/Water_density, ST *)
FUNCTION Water_density : REAL
VAR_INPUT
	T : REAL;
	Sat : BOOL;
END_VAR
VAR CONSTANT
	a0 : REAL := 999.83952;
	a1 : REAL := 16.952577;
	a2 : REAL := -7.9905127E-3;
	a3 : REAL := -4.6241757E-5;
	a4 : REAL := 1.0584601E-7;
	a5 : REAL := -2.8103006E-10;
	b  : REAL := 0.0168872;
END_VAR
VAR
	T2: REAL;
	T4: REAL;
END_VAR


(*
version 1.1	2 dec 2007
programmer 	hugo
tested by		tobias

this function calculates the water density for air free water between 0 and 100 deg C
while sat is false the denisty is calculated for air free water and when sat = true
the calculation is performed for water saturated with air.

*)
T2 := T * T;
T4 := T2 * T2;

(* original code changed for performance
Water_density := (a0 + a1*T + a2*EXPT(T,2) + a3*EXPT(t,3) + a4*EXPT(t,4) + a5*EXPT(t,5)) / (1 + b*T);
*)
Water_density := (a0 + a1*T + a2*T2 + a3*T2*T + a4*T4 + a5*T4*T) / (1 + b*T);

IF sat THEN Water_density := Water_density - 0.004612 + 0.000106 * T; END_IF;


(* revision history

hm	13.9.2007		rev 1.0
	original version

hm	2.12.2007		rev 1.1
	changed code for better performance
*)

(*
    °C - die Celsius-Temperatur in Grad Celsius
    v – das spezifische Volumen in Kubikdezimeter je Kilogramm dm³/kg
    h – die spezifische Enthalpie in Kilojoule je Kilogramm 	kJ/kg
    u – die spezifische Innere Energie in Kilojoule je Kilogramm 	kJ/kg
    s – die spezifische Entropie in Kilojoule je Kilogramm mal Kelvin 	kJ/(kg·K)
    cp - die spezifische Wärmekapazität bei konstantem Druck in Kilojoule je Kilogramm mal Kelvin 	kJ/(kg·K)
    Y – Volumenausdehnungskoeffizient in 10-3 durch Kelvin  10-3/K
    L – Wärmeleitfähigkeit in Milliwatt je Meter mal Kelvin  mW / (m·K) 
    n – Viskosität in Mikropascal mal Sekunde uPa·s 	
    s ? – Oberflächenspannung in Millinewton je Meter  mN/m


°C 		v 				h 			u 		s 			cp 		Y 		L		n		s	
-20		1,006580	
0 		1,000160 		0,06 		-0,04 	-0,0001 	4,228 	-0,080 	561,0 	1792 	75,65
4		1,000028
5 		1,0000 		21,1 		21,0 	0,076 		4,200 	0,011 	570,6 	1518 	74,95
10 		1,0003 		42,1 		42,0 	0,151 		4,188 	0,087 	580,0 	1306 	74,22
15 		1,0009 		63,0 		62,9 	0,224 		4,184 	0,152 	589,4 	1137 	73,49
20 		1,001797 		83,9 		83,8 	0,296 		4,183 	0,209 	598,4 	1001 	72,74
25 		1,0029 		104,8 		104,7 	0,367 		4,183 	0,259 	607,2 	890,4 	71,98
30 		1,0044 		125,8 		125,7 	0,437 		4,183 	0,305 	615,5 	797,7 	71,20
35 		1,0060 		146,7 		146,6 	0,505 		4,183 	0,347 	623,3 	719,6 	70,41
40 		1,007842 		167,58 	167,5 	0,572 		4,182 	0,386 	630,6 	653,3 	69,60
45 		1,0099 		188,5 		188,4 	0,638 		4,182 	0,423 	637,3 	596,3 	68,78
50 		1,0121 		209,4 		209,3 	0,704 		4,181 	0,457 	643,6 	547,1 	67,95
60 		1,017089 		251,2 		251,1 	0,831 		4,183 	0,522 	654,4 	466,6 	66,24
70 		1,0227 		293,1 		293,0 	0,955 		4,187 	0,583 	663,1 	404,1 	64,49
80 		1,029027 		335,0 		334,9 	1,075 		4,194 	0,640 	670,0 	354,5 	62,68
90 		1,0359 		377,0 		376,9 	1,193 		4,204 	0,696 	675,3 	314,6 	60,82
99,63 	1,0431 		417,5 		417,4 	1,303 		4,217 	0,748 	679,0 	283,0 	58,99
100	1,043453		419,1

Stoffdaten von Wasser Quelle Wickipedia

*)
END_FUNCTION

(* POU Building/HLK/water_enthalpy, ST *)
FUNCTION water_enthalpy : REAL
VAR_INPUT
	T : REAL;
END_VAR
VAR
	Pts : INT := 11;
	data : ARRAY[1..20, 0..1] OF REAL := 0,0.06, 10,42.1, 20,83.9, 30,125.8, 40,167.58, 50,209.4, 60,251.2, 70,293.1, 80,335.0, 90, 377.0, 100,419.1 ;
END_VAR

(*
version 1.0	29 oct 2007
programmer 	hugo
tested by		tobias

water_enthalpy calculates the enthalpy of liquid water from 0..100 °C 

*)
water_enthalpy := LINEAR_INT(T, Data, Pts);


(* revision history

hm	29.10.2007	rev 1.0
	original version

*)

(*
    °C - die Celsius-Temperatur in Grad Celsius
    v – das spezifische Volumen in Kubikdezimeter je Kilogramm dm³/kg
    h – die spezifische Enthalpie in Kilojoule je Kilogramm 	kJ/kg
    u – die spezifische Innere Energie in Kilojoule je Kilogramm 	kJ/kg
    s – die spezifische Entropie in Kilojoule je Kilogramm mal Kelvin 	kJ/(kg·K)
    cp - die spezifische Wärmekapazität bei konstantem Druck in Kilojoule je Kilogramm mal Kelvin 	kJ/(kg·K)
    Y – Volumenausdehnungskoeffizient in 10-3 durch Kelvin  10-3/K
    L – Wärmeleitfähigkeit in Milliwatt je Meter mal Kelvin  mW / (m·K) 
    n – Viskosität in Mikropascal mal Sekunde uPa·s 	
    s ? – Oberflächenspannung in Millinewton je Meter  mN/m


°C 		v 				h 			u 		s 			cp 		Y 		L		n		s	
-20		1,006580	
0 		1,000160 		0,06 		-0,04 	-0,0001 	4,228 	-0,080 	561,0 	1792 	75,65
4		1,000028
5 		1,0000 		21,1 		21,0 	0,076 		4,200 	0,011 	570,6 	1518 	74,95
10 		1,0003 		42,1 		42,0 	0,151 		4,188 	0,087 	580,0 	1306 	74,22
15 		1,0009 		63,0 		62,9 	0,224 		4,184 	0,152 	589,4 	1137 	73,49
20 		1,001797 		83,9 		83,8 	0,296 		4,183 	0,209 	598,4 	1001 	72,74
25 		1,0029 		104,8 		104,7 	0,367 		4,183 	0,259 	607,2 	890,4 	71,98
30 		1,0044 		125,8 		125,7 	0,437 		4,183 	0,305 	615,5 	797,7 	71,20
35 		1,0060 		146,7 		146,6 	0,505 		4,183 	0,347 	623,3 	719,6 	70,41
40 		1,007842 		167,58 	167,5 	0,572 		4,182 	0,386 	630,6 	653,3 	69,60
45 		1,0099 		188,5 		188,4 	0,638 		4,182 	0,423 	637,3 	596,3 	68,78
50 		1,0121 		209,4 		209,3 	0,704 		4,181 	0,457 	643,6 	547,1 	67,95
60 		1,017089 		251,2 		251,1 	0,831 		4,183 	0,522 	654,4 	466,6 	66,24
70 		1,0227 		293,1 		293,0 	0,955 		4,187 	0,583 	663,1 	404,1 	64,49
80 		1,029027 		335,0 		334,9 	1,075 		4,194 	0,640 	670,0 	354,5 	62,68
90 		1,0359 		377,0 		376,9 	1,193 		4,204 	0,696 	675,3 	314,6 	60,82
99,63 	1,0431 		417,5 		417,4 	1,303 		4,217 	0,748 	679,0 	283,0 	58,99
100	1,043453		419,1

Stoffdaten von Wasser Quelle Wickipedia

Wasser hat unter Normaldruck seine größte Dichte von 1000 Kilogramm pro Kubikmeter bei 3,98 °C und zeigt damit eine Dichteanomalie. 
Diese besteht darin, dass sich Wasser unterhalb von 3,98 °C bei weiterer Temperaturverringerung, auch beim Wechsel zum festen 
Aggregatzustand, wieder ausdehnt, was man nur von wenigen Stoffen kennt. Die derzeit genauesten publizierten Werte für die maximale 
Dichte liegen bei (999,974950 ± 0,00084) kg/m³ und bei (3,983 ± 0,00067) °C für die Temperatur, bei der dieser Wert erreicht wird. 
Die Werte stellen einen Mittelwert der von verschiedenen physikalischen Instituten veröffentlichten Zahlen dar (Stand 2001).

Die Berechnung der Dichte von luftfreiem Wasser DLF in Abhängigkeit von der Temperatur T ([T] = °C) kann mit Hilfe der folgenden 
Virialgleichung erfolgen:
: \frac{D_{\rm LF}}{\rm g/l} = \frac{a_0 + a_1 T + a_2 T^2 + a_3 T^3 + a_4 T^4 + a_5 T^5}{1 + b T}.
mit den Koeffizienten: a0 = 999,83952; a1 = 16,952577 (°C)-1; a2 = -7,9905127·10-3 (°C)-2; a3 = -4,6241757·10-5 (°C)-3; 
a4 = 1,0584601·10-7 (°C)-4; a5 = -2,8103006·10-10 (°C)-5 und b = 0,0168872. 
Für die Berechnung der Dichte von luftgesättigtem Wasser korrigiert man den Wert nach 
DLG/(g/l) = DLF/(g/l) - 0,004612 + 0,000106 (°C)-1·T. (Quelle: PTB-Mitteilungen 100/3-90)

*)
END_FUNCTION

(* POU mathematical/functions/LINEAR_INT, ST *)
FUNCTION LINEAR_INT : REAL
VAR_INPUT
	X : REAL;
	XY : ARRAY[1..20,0..1] OF REAL;
	Pts : INT;
END_VAR
VAR
	i : INT;
END_VAR

(*
	version 1.1	27 dec 2007
	programmer 	oscat
	tested BY		oscat

LINEAR_INT calculates an output based on a linear interpolation of up to 20 coordinates given in an array
the input coordinates have to start at the lowest array position and must be sorted ba ascending X values.

*)
(*make sure n is bound within the array size *)
pts := MIN(pts,20);

(* calculate the linear segement interpolation *)
i := 2;
(* search for segment and calculate output
	below and above the defined segments we interpolate the last segment *)
WHILE (i < pts) AND (XY[i,0] < X) DO
	i := i + 1;
END_WHILE;

(* calculate the output value on the corresponding segment coordinates *)
LINEAR_INT := ((XY[i,1] - XY[i-1,1]) * X - XY[i,1] * XY[i-1,0] + XY[i-1,1]*XY[i,0]) / (XY[i,0] - XY[i-1,0]);

(* revision history
hm	7. oct 2007		rev 1.0
	original version

hm	27 dec 2007		rev 1.1
	changed code for better performance
*)
END_FUNCTION

(* POU Building/HLK/Heat_temp, ST *)
FUNCTION_BLOCK Heat_temp
VAR_INPUT
	T_ext : REAL;
	Offset : REAL;
	t_req : REAL;
END_VAR
VAR_INPUT CONSTANT
	TY_max : REAL := 70;
	TY_min : REAL := 20;
	T_int : REAL := 20;
	TY_config : REAL := 50;
	T_ext_config : REAL := -15;
	C : REAL := 1.33;
END_VAR
VAR_OUTPUT
	Ty : REAL;
END_VAR
VAR
END_VAR

(*
version 1.0	27 jan 2007
programmer 	hugo
tested by		tobias

Heat_Temp calculates a heat characteristic based on the formula: tv=ti+(tvmax-ti)*((ti-tau)/(ti-taumin))^(1/n)
while
tv necessary heating temperature.
ti internal room temperature (20°C)
tau current external temperature
external temperature to determine characteristics
C exponent for heating system (normally 1,33 or 1,1 for floor heating)

The two additional inputs TY_min and TY_max set limits for the output TY, while an offset inputs allows to rise or lower the room temperature.

*)
IF t_ext > t_int + Offset THEN
	ty := t_int + offset;
ELSE
Ty := T_int - offset + (TY_config - T_int) * EXPT((T_int - offset - T_ext) / (T_int - offset - T_ext_config),1 / C);
END_IF;
IF t_req > ty THEN ty := t_req; END_IF;
ty := LIMIT(TY_min, ty, TY_max);



(*

tv=ti+(tvmax-ti)*((ti-tau)/(ti-taumin))^(1/n)

tv aktuelle Vorlauftemp.
ti Raumtemperatur innen (20°C)
tau aktuelle Außentemperatur
taumin minimale Außentemperatur -12°C oder -15°C
n Heizkörperexponent (meistens 1,33)
Fußbodenheizung = 1,1
Wandheizung 1,3

Normen z. B. DIN 4703, DIN 4725 oder die Literatur, z. B Recknagel Abschnitt 1.3.5.

*)
END_FUNCTION_BLOCK

(* POU Building/HLK/legionella, ST *)
FUNCTION_BLOCK legionella
VAR_INPUT
	manual : BOOL;
	temp_boiler : REAL;
	temp_return : REAL := 100;
	DT_in: DT;
	rst : BOOL;
END_VAR
VAR_INPUT CONSTANT
	T_start: TOD := tod#03:00:00;
	day : INT := 7;
	temp_set : REAL := 70;
	temp_offset : REAL := 10;
	temp_hys : REAL := 5;
	t_max_heat: TIME := t#10m;
	t_max_ret : TIME := t#10m;
	tp_0: TIME := t#5m;
	tp_1: TIME := t#5m;
	tp_2: TIME := t#5m;
	tp_3: TIME := t#5m;
	tp_4: TIME := t#5m;
	tp_5: TIME := t#5m;
	tp_6: TIME := t#5m;
	tp_7: TIME := t#5m;
END_VAR
VAR_OUTPUT
	Heat : BOOL;
	pump : BOOL;
	valve0 : BOOL;
	valve1 : BOOL;
	valve2 : BOOL;
	valve3 : BOOL;
	valve4 : BOOL;
	valve5 : BOOL;
	valve6 : BOOL;
	valve7 : BOOL;
	run: BOOL;
	Status : BYTE;
END_VAR
VAR
	X1: timer_1;
	x2: sequence_8;
	x3: hyst_1;
	init: BOOL;
END_VAR

(*
version 1.1	17. jan 2007
programmer 	oscat
tested by		hans

Legionella is a complete sequencer for up to 8 hot water lines that need to be sterilzed periodically.
legionella needs a DT input with the appropriate time, usually gererated by the rtc of the system. for system independence this time is connected externally.
T_start is the time when sterilazation should be started and day is the day_of_week when it should be performed (1=Monday and 7=sunday).
so sterilazation is autioimatically performed once a week at a specified time.
temp_set and temp_hys and temp_offset specify the boiler temperatur nedded for sterilization. as a defaut Temp_set is set to 70 deg C and Temp_hys is set to 5 deg C and temp_offset is 10 deg C.
a temp boiler input reads the boiler temperature of the hot water tank.
after a start pulse is gererated by the weekly timer or a manual test input the sequence is started:
1. the boiler is heated to temp_set + temp_offset + temp_hys = 85 deg C unless chaged at setup.
	the heat output is turned on and tells the heater to turn heating on. if the temp is not reached for a time of t_max_heat (10 min) the error output is set and the sequence is stopped.
2. after the specified temperature is reached, the output valve0 and pump is turned on and starts sterilization of line0 until temp_return has reached temp_set and continues to sterilize for a time of tp_0 (5 min default).
	if tmep_set is not reached at the temp_return_input then the error output is set and the sequence will be stopped.
	if there is no temp sensor for temp_return (the temperature at the return point for the circulation pump pls set this imput to a value greater then temp_set (by default use 100 deg C).
	in this case sterilization is performed for the default times without monitoring the return temp.
3. this sequence is repeated for up to valves.

connection scheme:

temp_boiler:	input oif the boiler temperature sensor.
temp_hys:		config value for the heater hysteresis, preset to 5 deg C.
temp_offset:	config value for the heater temp_offset against temp_set, preset to 10 deg C.
temp_set:		config value for the specified sterilization temperature, preset to 70 deg C.
temp_return:	input of the circulation return line temperature sensor, if not availabe set this value to 100 deg C.
manual:		manual input to start the sterilization by hand for diagnostic purposes, rising edge active, leave low for automatic operation.
DT_in:			date,time input supplied by a external real time clock.
T_start:		time of day when the sterilization should be started.
day:			config value for day of week when the process should be started, preset to sunday.
t_max_hest:	tmax time to be needed for the heater to heat the hot water tank to the specified value, preset to 10 min.

*)
(* startup initialization *)
IF NOT init THEN
	init := TRUE;
	X1.start_day := day;
	X1.start_time := T_start;
	X3.low := Temp_offset + temp_set;
	X3.high := Temp_hys + X3.low;
	X2.wait0 := T_max_heat;
	X2.delay0 := TP_0;
	X2.delay1 := TP_1;
	X2.delay2 := TP_2;
	X2.delay3 := TP_3;
	X2.delay4 := TP_4;
	X2.delay5 := TP_5;
	X2.delay6 := TP_6;
	X2.delay7 := TP_7;
	X2.wait1 := T_max_ret;
	X2.wait2 := T_max_ret;
	X2.wait3 := T_max_ret;
	X2.wait4 := T_max_ret;
	X2.wait5 := T_max_ret;
	X2.wait6 := T_max_ret;
	X2.wait7 := T_max_ret;
	X2();
END_IF;

(* oerational code *)
X1(DT_in := DT_in);
IF X1.Q OR manual OR x2.run THEN
	X3(in := temp_boiler);
	X2.in0 := X3.Q OR x3.win;
	X2.in1 := temp_return >= temp_set;
	X2.in2 := x2.in1;
	X2.in3 := x2.in1;
	X2.in4 := x2.in1;
	X2.in5 := x2.in1;
	X2.in6 := x2.in1;
	X2.in7 := x2.in1;
	X2.rst := rst;
	X2(start := X1.Q OR manual);
	run := x2.run;
	pump := x2.any;
	Heat := NOT X3.Q AND x2.run;
	valve0 := X2.Q0;
	valve1 := X2.Q1;
	valve2 := X2.Q2;
	valve3 := X2.Q3;
	valve4 := X2.Q4;
	valve5 := X2.Q5;
	valve6 := X2.Q6;
	valve7 := X2.Q7;
	pump := X2.any;
	status := X2.status;
ELSE;
	X2(start :=0);
	status := x2.status;
END_IF;

(* revision history

hm 17.jan 2007	rev 1.1
	rewritten to st for higher performance
	changes eeror output to esr compatible status output
*)
END_FUNCTION_BLOCK

(* POU Logic/generators/sequence_8, ST *)
FUNCTION_BLOCK sequence_8
VAR_INPUT
	in0 : BOOL := TRUE;
	in1 : BOOL := TRUE;
	in2 : BOOL := TRUE;
	in3 : BOOL := TRUE;
	in4 : BOOL := TRUE;
	in5 : BOOL := TRUE;
	in6 : BOOL := TRUE;
	in7 : BOOL := TRUE;
	start : BOOL;
	rst : BOOL;
	wait0 : TIME := t#0s;
	delay0 : TIME := t#0s;
	wait1 : TIME := t#0s;
	delay1 : TIME := t#0s;
	wait2 : TIME := t#0s;
	delay2 : TIME := t#0s;
	wait3 : TIME := t#0s;
	delay3 : TIME := t#0s;
	wait4 : TIME := t#0s;
	delay4 : TIME := t#0s;
	wait5 : TIME := t#0s;
	delay5 : TIME := t#0s;
	wait6 : TIME := t#0s;
	delay6 : TIME := t#0s;
	wait7 : TIME := t#0s;
	delay7 : TIME := t#0s;
END_VAR
VAR_INPUT CONSTANT
	stop_on_error : BOOL := FALSE;
END_VAR
VAR_OUTPUT
	Q0 : BOOL;
	Q1 : BOOL;
	Q2 : BOOL;
	Q3 : BOOL;
	Q4 : BOOL;
	Q5 : BOOL;
	Q6 : BOOL;
	Q7 : BOOL;
	any : BOOL;
	run: BOOL;
	step : INT := -1;
	status : BYTE;
END_VAR
VAR
	last : TIME;
	edge : BOOL;
	tx: TIME;
	init: BOOL;
END_VAR

(*
version 1.4	17 sep 2007
programmer 	oscat
tested by		hans

